	(* ----------------------------------------------------------------------------
	Const name  : FSM_EVENT_ARRAY_MAX
	Description : Max event array index value in the FSM table
				  Must subtract 1 due to arrays starting at 0
	Notes       : Used in FSM table definitions
	---------------------------------------------------------------------------- *)
	FSM_EVENT_ARRAY_MAX: INT := FSM_NUM_EVENTS - 1;
	
	(* ----------------------------------------------------------------------------
	Const name  : FSM_ACTIONS_ARRAY_MAX
	Description : Max actions array index value in the FSM table
				  next state entry is element 0 
	Notes       : Used in FSM table definitions
	---------------------------------------------------------------------------- *)
	FSM_ACTIONS_ARRAY_MAX: INT := FSM_NUM_EVENT_ACTIONS;

END_VAR

// (* FSM *)

//Run the Tri State Valve Finite State Machine Logic Block <JAISON>
m_TriStateValveControlFSM(xEnable:= xEnable, xError=> m_FsmError, errorNum=> m_FsmErrorNum);

//Set the current FSM State variable for testing the FSM state transitions <JAISON>
m_FsmCurrentState := m_TriStateValveControlFSM.FSM_GetCurrentState();

// Run the valve shift timer, the timer is enabled/disabled in the action handler. <JAISON>
//m_ShiftTimer(IN:= (m_TriStateValveControlFSM.FSM_GetCurrentState() = TriStateValveFsmState.FsmState_ValveShifting), PT:= ValveShiftTimeout);
m_ShiftTimer(PT:= ValveShiftTimeout);

// (* VALVE FEEDBACK *)
// Determine the current valve state (position) based on the feedback <JAISON>

// If the open and closed feedback are both TRUE or both FALSE the valve position is unknown
IF (Opened_Feedback = Closed_Feedback) THEN
	
	ValvePosition := TValveTriStatePosition.PosUnknown;
	
// If the opened feedback is TRUE and closed feedback is FALSE then the valve is opened
ELSIF ((Opened_Feedback) AND (NOT Closed_Feedback)) THEN
	
	ValvePosition := TValveTriStatePosition.PosOpened;
	
// If the closed feedback is TRUE and the open feedback is FALSE then the valve is closed
ELSIF ((Closed_Feedback) AND (NOT Opened_Feedback)) THEN
	
	ValvePosition := TValveTriStatePosition.PosClosed;
	
END_IF

// (* EVENT TRIGGERS *)

// Valve enabled trigger, basic FSM Event with no user parameters <JAISON>
m_EnableTrigger(CLK:= xEnable);
IF (m_EnableTrigger.Q)THEN
	//  FSM Reset needs to be called outside of the Action Handler routine. 
	//	Reset the FSM before sending the enable event. <JAISON>
	m_TriStateValveControlFSM.FSM_Reset();
	m_TriStateValveControlFSM.FSM_ProcessEvent(event:= TriStateValveFsmEvent.FsmEvent_ValveEnable);
END_IF

// Valve disabled trigger, basic FSM Event with no user parameters <JAISON>
m_DisableTrigger(CLK:= xEnable);
IF (m_DisableTrigger.Q)THEN
	m_TriStateValveControlFSM.FSM_ProcessEvent(event:= TriStateValveFsmEvent.FsmEvent_ValveDisable);
END_IF

// Valve shift timeout expired event trigger, basic FSM Event with no user parameters <JAISON>
m_ShiftTimeoutTrigger(CLK:= m_ShiftTimer.Q);
IF (m_ShiftTimeoutTrigger.Q) THEN
	m_TriStateValveControlFSM.FSM_ProcessEvent(event:= TriStateValveFsmEvent.FsmEvent_ValveShiftTimerExpired);
END_IF

// Valve opened event trigger, basic FSM Event with no user parameters <JAISON>
m_OpenedTrigger(CLK:= (ValvePosition = TValveTriStatePosition.PosOpened) AND (m_ValveCmdPosition = TValveTriStatePosition.PosOpened));
IF (m_OpenedTrigger.Q) THEN
	m_TriStateValveControlFSM.FSM_ProcessEvent(event:= TriStateValveFsmEvent.FsmEvent_ValveOpened);
END_IF

// Valve closed event trigger, basic FSM Event with no user parameters <JAISON>
m_ClosedTrigger(CLK:= (ValvePosition = TValveTriStatePosition.PosClosed) AND (m_ValveCmdPosition = TValveTriStatePosition.PosClosed));
IF (m_ClosedTrigger.Q) THEN
	m_TriStateValveControlFSM.FSM_ProcessEvent(event:= TriStateValveFsmEvent.FsmEvent_ValveClosed);
END_IF

// Valve position mismatch event trigger, basic FSM Event with no user parameters <JAISON>
// <Note: Ensure the cmd position is valid before sending event, this means valve has been shifted AT LEAST once.> <JAISON>
m_PositionMismatchTrigger(CLK:= ((m_ValveCmdPosition <> ValvePosition) AND ((m_ValveCmdPosition = TValveTriStatePosition.PosOpened) OR (m_ValveCmdPosition = TValveTriStatePosition.PosClosed))));
IF (m_PositionMismatchTrigger.Q) THEN
	m_TriStateValveControlFSM.FSM_ProcessEvent(event:= TriStateValveFsmEvent.FsmEvent_ValvePositionMismatch);
END_IF

(* ---------------------------------------------------------------------------
Func name   : 	CloseValve
Description : 	Sends an valve close event the the FSM 
				if the block is Enabled.
Inputs      :	None
Returns     : 	None
Notes       : 	This method should be triggered by an event 
				and not called cyclically to prevent flooding 
				the FSM event Queue.
--------------------------------------------------------------------------- *)

METHOD CloseValve : BOOL
VAR_INPUT
END_VAR
// Send the valve open event if the valve is enabled
IF xEnable THEN
	
	// Reset the valve shift timeout timer
	m_ShiftTimer(IN:= FALSE);
		
	// Clear the shifting error output
	ShiftingError := FALSE;

	m_TriStateValveControlFSM.FSM_ProcessEvent(event:= TriStateValveFsmEvent.FsmEvent_ValveClose);
	
END_IF
END_METHOD

(* ---------------------------------------------------------------------------
Func name   : 	ExecuteAction
Description : 	This method is a standardized handler for
				each action generated by the FSM
Inputs      :	p_FSM			-	pointer to the instantiation of the FSM object
				currentAction	-	current FSM action being processed
				currentEvent	-	current FSM event being processed
Returns     : 	BOOL			- 	result of action function (returning true means change state)
Notes       : 	The approach of using an interface enables the user 
				of the FSM to define and handle actions based 
				on their design and implementation.
				
				Return TRUE to change state, FALSE to remain in 
				the same state, unless the FSM has the alwaysChangeState
				set to TRUE, then it will change state regardless 
				of action handler return.
				
				If a conditional state is to be used this action handler
				routuine is responsible for setting the conditionalState 
				value using the FSM_SetConditionalState() function.
--------------------------------------------------------------------------- *)

METHOD ExecuteAction : BOOL
VAR_INPUT
	p_FSM			: POINTER TO fb_FSM;			// Pointer to the instantiation of the FSM object
	currentAction	: TFsmAction;					// Current FSM action being processed
	currentEvent	: TFsmEventDesc;				// Current FSM event being processed
END_VAR
VAR_OUTPUT

END_VAR
VAR

END_VAR
CASE currentAction OF
	
	TriStateValveFsmAction.FsmAction_None:
		
		// DO ACTION NONE
			
		// This would be a good place to simply log that the event occured. <JAISON>
			
		// RETURN TRUE
		ExecuteAction := TRUE;
	
	TriStateValveFsmAction.FsmAction_ValveEnabled:
	
		// DO ACTION VALVE ENABLED

		// Disable the actuator outputs
		Open_Actuator := FALSE;	
		Close_Actuator := FALSE;

		// Clear the shifting error to FALSE
		ShiftingError := FALSE;

		// Reset the valve shift timer
		m_ShiftTimer(IN := FALSE);

		// Clear all event triggers to ensure all events are captured on startup
		// NOTE: DO NOT RESET ENABLE/DISABLE TRIGGERS <JAISON>
		m_OpenedTrigger(CLK:= FALSE);
		m_ClosedTrigger(CLK:= FALSE);
		m_PositionMismatchTrigger(CLK:= FALSE);
		m_ShiftTimeoutTrigger(CLK:= FALSE);

		// Shift the valve to the Initial Valve State
		CASE InitialValvePosition OF
			
			TValveTriStatePosition.PosOpened:
			
				OpenValve();
			
			TValveTriStatePosition.PosClosed:
			
				CloseValve();
				
		ELSE
		
			// Error - Retained valve position invalid  <MESSAGE>
			// Default to CLOSED <JAISON>
			CloseValve();
		
		END_CASE
		
		// RETURN TRUE
		ExecuteAction := TRUE;
		
	TriStateValveFsmAction.FsmAction_ValveDisabled:	

		// DO ACTION VALVE DISABLED
		
		// Disable the actuator outputs
		Open_Actuator := FALSE;	
		Close_Actuator := FALSE;
		
		// RETURN TRUE
		ExecuteAction := TRUE;
		
	TriStateValveFsmAction.FsmAction_ValveOpen:
		
		// DO ACTION VALVE OPEN
		
		// Enable the Open actuator and Disable the Close actuator
		Close_Actuator := FALSE;
		Open_Actuator := TRUE;
		
		// Set the desired valve position to OPEN
		m_ValveCmdPosition := TValveTriStatePosition.PosOpened;
		
		// Start the valve shift timeout timer
		m_ShiftTimer(IN:= TRUE);
		
		// RETURN TRUE
		ExecuteAction := TRUE;
			
	TriStateValveFsmAction.FsmAction_ValveClose:
		
		// DO ACTION VALVE CLOSE

		// Enable the Close actuator and Disable the Open actuator
		Open_Actuator := FALSE;
		Close_Actuator := TRUE;
		
		// Set the desired valve position to CLOSE
		m_ValveCmdPosition := TValveTriStatePosition.PosClosed;
		
		// Start the valve shift timeout timer
		m_ShiftTimer(IN:= TRUE);
		
		// RETURN TRUE
		ExecuteAction := TRUE;
			
	TriStateValveFsmAction.FsmAction_ValveOpened:
		
		// DO ACTION VALVE OPENED
		
		// Disable both the Open and Close actuators
		Open_Actuator := FALSE;
		Close_Actuator := FALSE;
		
		// Clear the shifting error output
		ShiftingError := FALSE;
		
		// Stop the valve shift timeout timer
		m_ShiftTimer(IN:= FALSE);
		
		// RETURN TRUE
		ExecuteAction := TRUE;
			
	TriStateValveFsmAction.FsmAction_ValveClosed:
		
		// DO ACTION VALVE CLOSED
			
		// Disable both the Open and Close actuators
		Open_Actuator := FALSE;
		Close_Actuator := FALSE;
		
		// Clear the shifting error output
		ShiftingError := FALSE;
		
		// Stop the valve shift timeout timer
		m_ShiftTimer(IN:= FALSE);
		
		// RETURN TRUE
		ExecuteAction := TRUE;
			
	TriStateValveFsmAction.FsmAction_ValveShiftTimerExpired:
		
		// DO ACTION VALVE SHIFT TIMER EXPIRED
	
		// Set the shifting error output
		ShiftingError := TRUE;
				
		// RETURN TRUE
		ExecuteAction := TRUE;
		
	TriStateValveFsmAction.FsmAction_ValvePositionMismatch:
		
		// DO ACTION VALVE POSITION MISMATCH
		
		CASE m_ValveCmdPosition OF
			TValveTriStatePosition.PosOpened:
			
				// If the desired valve position is to be opened and the valve drifted then activate the open command again.
				p_FSM^.FSM_ProcessEvent(event:= TriStateValveFsmEvent.FsmEvent_ValveOpen);
			
			TValveTriStatePosition.PosClosed:
			
				// If the desired valve position is to be closed and the valve drifted then activate the close command again.
				p_FSM^.FSM_ProcessEvent(event:= TriStateValveFsmEvent.FsmEvent_ValveClose);
			
			ELSE
				
				// Error - Desired position unknown - Should not happen
				// NOTE: 	This will HALT the FSM when it FAILS which might not be the desired behavior.
				//			It is NOT necessary to halt the FSM, instead an unexpected event might just
				//			place the FSM into an error state which will allow actions to be ran. <JAISON>
				p_FSM^.FSM_ASSERT(FALSE, TFsmError.FSM_INVALID_EVENT_ERROR);
				
		END_CASE
		
		// RETURN TRUE
		ExecuteAction := TRUE;
			
	FSM_ACTION_UNEXPECTED_EVENT:
		
		// DO ACTION UNEXPECTED EVENT
		
		// ERROR TRAP - UNKNOWN ACTION
		// NOTE: 	This will HALT the FSM when it FAILS which is likely advisable here because
		//			this is a critical design time error.  All actions need to be defined, even
		//			if they simply log an event occured. <JAISON>
		p_FSM^.FSM_ASSERT(FALSE, TFsmError.FSM_INVALID_ACTION);
		
		// RETURN FALSE
		ExecuteAction := FALSE;
		
	FSM_ACTION_ERROR_EVENT:
	
		// DO ACTION ERROR EVENT
		
		// This action is executed when an FSM ASSERT Fails and the FSM is transitioning to the defined error state. <JAISON>
		
		// Automatically Reset the Valve / FSM by toggling the enable which will force the FSM to reset to Valve Off state
		m_EnableTrigger(CLK:= FALSE);
		
		// RETURN FALSE - This is irrelevant because the FSM will automatically transition to the error state.
		ExecuteAction := FALSE;
			
ELSE
		
	// ERROR TRAP - UNKNOWN ACTION
	// NOTE: 	This will HALT the FSM when it FAILS which is likely advisable here because
	//			this is a critical design time error.  All actions need to be defined, even
	//			if they simply log an event occured. <JAISON>
	p_FSM^.FSM_ASSERT(FALSE, TFsmError.FSM_INVALID_ACTION);
		
	// RETURN FALSE
	ExecuteAction := FALSE;
		
END_CASE;

m_FsmLastEvent := currentEvent.event;
m_FsmLastAction := currentAction;
m_FsmLastState := p_FSM^.FSM_GetPreviousState();
END_METHOD

(* ---------------------------------------------------------------------------
Func name   : 	FB_exit
Description : 	Destructor
Inputs      :	None
Returns     : 	None
Notes       : 	
--------------------------------------------------------------------------- *)

METHOD FB_exit : BOOL
VAR_INPUT
	bInCopyCode : BOOL; // if TRUE, the exit method is called for exiting an instance that is copied afterwards (online change)
END_VAR
// Do nothing
END_METHOD

(* ---------------------------------------------------------------------------
Func name   : 	FB_init
Description : 	Constructor
Inputs      :	None
Returns     : 	None
Notes       : 	
--------------------------------------------------------------------------- *)

METHOD FB_init : BOOL
VAR_INPUT
	bInitRetains 		: BOOL; 				// if TRUE, the retain variables are initialized (warm start / cold start)
    bInCopyCode  		: BOOL; 				// if TRUE, the instance afterwards gets moved into the copy code (online change)
END_VAR
// Set the FSM error state
// Technically this valve does NOT use the error state as it just resets itself 
// on transition to this state, however it is a good practice to have and will
// be useful for other state machines. <JAISON>
m_TriStateValveControlFSM.FSM_SetErrorState(TriStateValveFsmState.FsmState_Error);

// Clear all event triggers to ensure all events are captured on startup
m_EnableTrigger(CLK:= FALSE);
m_DisableTrigger(CLK:= FALSE);
m_OpenedTrigger(CLK:= FALSE);
m_ClosedTrigger(CLK:= FALSE);
m_PositionMismatchTrigger(CLK:= FALSE);
m_ShiftTimeoutTrigger(CLK:= FALSE);

// Initialize the default valve cmd state to unknown as this will be properly set during the valve enable. <JAISON>
m_ValveCmdPosition := TValveTriStatePosition.PosUnknown;

// Disable the actuator outputs
Open_Actuator := FALSE;	
Close_Actuator := FALSE;

// Initialize the shifting error to FALSE
ShiftingError := FALSE;
END_METHOD

(* ---------------------------------------------------------------------------
Func name   : 	OpenValve
Description : 	Sends an valve open event the the FSM 
				if the block is Enabled.
Inputs      :	None
Returns     : 	None
Notes       : 	This method should be triggered by an event 
				and not called cyclically to prevent flooding 
				the FSM event Queue.
--------------------------------------------------------------------------- *)

METHOD OpenValve
VAR_INPUT
END_VAR
// Send the valve open event if the valve is enabled
IF xEnable THEN

	// Reset the valve shift timeout timer
	m_ShiftTimer(IN:= FALSE);
		
	// Clear the shifting error output
	ShiftingError := FALSE;	

	m_TriStateValveControlFSM.FSM_ProcessEvent(event:= TriStateValveFsmEvent.FsmEvent_ValveOpen);
	
END_IF
END_METHOD

END_FUNCTION_BLOCK

// 20 Program Organization Units/Equipment Functions/TriStateValve/fb_DigitalFeedbackDualActionValve
(*AUTHOR:			Ryan Herdian*)
(*DATE:				July 30, 2020*)
(*DESCRIPTION: 		This function block provides the functionality for a Tri-State dual action valve which
					has digital boolean Open/Close feedback.  This valve is controlled by output
					boolean Open/Close solenoid and motor.*)

(*NOTES:			Operation of the valve are to follow
					To Open:
					-	Energize both solenoid and motor output at the same time. Until open. 
					-	Leave about 5 seconds after in position
					-	Remove power
					
					To Close:
					-	Energize the motor output only until close
					-	Leave about 5 seconds
					-	Remove power
					
					Currently, this function block is intended for
					- Emerson Damcos LPU-D
*)

(*UPDATE: 			March. 23 2021 - Jaison Schaab

					Code Is fully tested and functional.				
*)

(*UPDATE: 			March. 18 2021 - Jaison Schaab

					Code Ported from Wago.
					
					Code has NOT Yet been tested.
*)
	
(*UPDATE: 			September. 3 2020 - Jaison Schaab

					Added a "IsShifting" method for use in the control class development to detect when valve is shifting.
*)
					
(*UPDATE: 			September. 1 2020 - Jaison Schaab

					Added a "IsShiftingError" method for use in the control class development to detect valve shift error.
					
					Moved the setting of the outputs to occur through triggers rather than in the methods.  This was because
					during testing of the suction control class I noticed that the valves would not initially shift the their
					default position on startup; which is a massive concern.
*)

FUNCTION_BLOCK fb_DigitalFeedbackDualActionValve
VAR_INPUT
	xEnable						: BOOL;						// Enable inputs and valve operation
	OpenCommand					: BOOL;						// Open valve command input
	CloseCommand				: BOOL;						// Close valve command input
	InitialValvePosition		: TValveTriStatePosition;	// Position the valve will shift to when enabled (To be retianed if desired outside this block)
	OpenedFeedback				: BOOL;						// Digital feedback (TRUE = valve OPENED)
	ClosedFeedback				: BOOL;						// Digital feedback (TRUE = valve CLOSED)
	ValveShiftTimeout			: TIME;						// Valve shift timout value
	ValveOutputDisableTime		: TIME;						// Time to disable the output after shifting 
END_VAR
VAR_OUTPUT
	ValvePosition				: TValveTriStatePosition;	// Current valve position	(0 = closed, 1 = open)
	SolenoidEnergized			: BOOL;								// Solenoid energized (TRUE to OPEN valve together with Motor)
	MotorEnergized				: BOOL;								// Motor energized (TRUE to OPEN valve together with Solenoid)
END_VAR
VAR
	(* TriState Valve Function Block *)	

	m_TriStateValve				: fb_TriStateValve;			// Tri-State valve common control with state machine
	
	(* Valve Status *)	
	m_OpenedFeedback			: BOOL;						// Internal valve opened feedback
	m_ClosedFeedback			: BOOL;						// Internal valve closed feedback
	
	m_ValveShiftError			: BOOL;						// Valve shift timeout error flag
	
	(* Valve Internal Command *)
	m_OpenActuator				: BOOL;						// Internal Valve open actuator (TRUE to OPEN valve)
	m_CloseActuator				: BOOL;						// Internal Valve close actuator (TRUE to CLOSE valve)
	
	(* Alarms *)
	m_ValveShiftTimeout			: fb_AlarmMonitor;			// Alarm monitor for valve shift timeout error
	
	(* Event Triggers *)	

	m_EnableTrigger				: R_TRIG;					// Valve enabled trigger
	m_DisableTrigger			: F_TRIG;					// Valve disabled trigger
	m_OpenTrigger				: R_TRIG;					// Valve open trigger
	m_CloseTrigger				: R_TRIG;					// Valve close trigger
	m_ValveShiftErrorTrigger	: R_TRIG;					// Valve shift error trigger
	
	m_SetOpenActuatorTrigger	: R_TRIG;					// Set open actuator trigger
	m_SetCloseActuatorTrigger	: R_TRIG;					// Set close actuator trigger
	
	m_DisableOutputTrigger		: R_TRIG;					// Disable output trigger
	
	
	// ---- move this to the appropriate section
	//m_ValveShifted				: BOOL;
	// ----
	
	(* TIMER *)
	m_ValveShiftedTimer			: TON;
	
END_VAR

// Run the common TriState Valve function block which manages the state machine
m_TriStateValve(	xEnable					:= xEnable, 
					InitialValvePosition	:= InitialValvePosition,
					Opened_Feedback			:= m_OpenedFeedback, 
					Closed_Feedback			:= m_ClosedFeedback, 
					ValveShiftTimeout		:= ValveShiftTimeout,
					ValvePosition			=> ValvePosition, 
					Open_Actuator			=> m_OpenActuator, 
					Close_Actuator			=> m_CloseActuator, 
					ShiftingError			=> m_ValveShiftError);
					

(* TIMER *)
m_ValveShiftedTimer(IN:= IsOpened() OR IsClosed(), PT:= ValveOutputDisableTime);


// (* EVENT TRIGGERS *)

// Valve enabled trigger
m_EnableTrigger(CLK:= xEnable);
IF (m_EnableTrigger.Q)THEN
	
	// De-energized the Solenoid and Motor
	SolenoidEnergized := FALSE;
	MotorEnergized := FALSE;

	// Disable the internal actuator outputs
	m_OpenActuator := FALSE;	
	m_CloseActuator := FALSE;

	// Clear all event triggers to ensure all events are captured on startup
	// NOTE: DO NOT RESET ENABLE/DISABLE TRIGGERS
	m_OpenTrigger(CLK:= FALSE);
	m_CloseTrigger(CLK:= FALSE);
	
	m_ValveShiftErrorTrigger(CLK:= FALSE);
	
	m_SetOpenActuatorTrigger(CLK:= FALSE);
	m_SetCloseActuatorTrigger(CLK:= FALSE);
	
END_IF

// Valve disabled trigger
m_DisableTrigger(CLK:= xEnable);
IF (m_DisableTrigger.Q)THEN
	// Disable the alarm monitor
	m_ValveShiftTimeout.DisableLimit();
END_IF

// Open valve command event trigger
m_OpenTrigger(CLK:= OpenCommand);
IF (m_OpenTrigger.Q) THEN	
	OpenValve();	
END_IF

// Close valve command event trigger
m_CloseTrigger(CLK:= CloseCommand);
IF (m_CloseTrigger.Q) THEN
	CloseValve();		
END_IF

// Valve shift error event trigger
m_ValveShiftErrorTrigger(CLK:= m_ValveShiftError);
IF (m_ValveShiftErrorTrigger.Q) THEN
	// Reset the open/close actuator triggers to reissue the last command outputs
	m_SetOpenActuatorTrigger(CLK:= FALSE);
	m_SetCloseActuatorTrigger(CLK:= FALSE);
END_IF

// Open acutator trigger
m_SetOpenActuatorTrigger(CLK:= m_OpenActuator);
IF (m_SetOpenActuatorTrigger.Q) THEN
	SolenoidEnergized	:= TRUE;
	MotorEnergized		:= TRUE;
END_IF

// Close actuator trigger
m_SetCloseActuatorTrigger(CLK:= m_CloseActuator);
IF (m_SetCloseActuatorTrigger.Q) THEN
	MotorEnergized 		:= TRUE;
	SolenoidEnergized 	:= FALSE;		
END_IF
	
// Disable Output Trigger
m_DisableOutputTrigger(CLK:= m_ValveShiftError OR m_ValveShiftedTimer.Q);
IF (m_DisableOutputTrigger.Q)THEN	
	// De-energized the Solenoid and Motor
	SolenoidEnergized 	:= FALSE;
	MotorEnergized 		:= FALSE;	
END_IF


// (* VALVE FEEDBACK *)

// Decode the valve feedback
m_OpenedFeedback := OpenedFeedback;
m_ClosedFeedback := ClosedFeedback;


// Run the Alarm Monitors
m_ValveShiftTimeout.MonitorBool(value:= m_ValveShiftError);

(* ---------------------------------------------------------------------------
Func name   : 	CloseValve
Description : 	Sends an valve close event the the Tri-State valve if the block is Enabled.
				De-energize the Solenoid and Energize the Motor to close the valve if the
				valve has not already in the closed position.
Inputs      :	None
Returns     : 	None
Notes       : 	This method should be triggered by an event 
				and not called cyclically to prevent flooding 
				the FSM event Queue.
--------------------------------------------------------------------------- *)

METHOD CloseValve : BOOL
VAR_INPUT
END_VAR
// Send CLOSE command to Tri-State Valve FSM if the valve is enabled
IF xEnable THEN
	m_TriStateValve.CloseValve();	
END_IF
END_METHOD

(* ---------------------------------------------------------------------------
Func name   : 	FB_exit
Description : 	Destructor
Inputs      :	None
Returns     : 	None
Notes       : 	
--------------------------------------------------------------------------- *)

METHOD FB_exit : BOOL
VAR_INPUT
	bInCopyCode : BOOL; // if TRUE, the exit method is called for exiting an instance that is copied afterwards (online change)
END_VAR
// Do Nothing
END_METHOD

(* ---------------------------------------------------------------------------
Func name   : 	FB_init
Description : 	Constructor
Inputs      :	None
Returns     : 	None
Notes       : 	
--------------------------------------------------------------------------- *)

METHOD FB_init : BOOL
VAR_INPUT
	bInitRetains 		: BOOL; 				// if TRUE, the retain variables are initialized (warm start / cold start)
    bInCopyCode  		: BOOL; 				// if TRUE, the instance afterwards gets moved into the copy code (online change)
END_VAR
// Disable the solenoid and motor outputs
SolenoidEnergized := FALSE;
MotorEnergized := FALSE;

// Disable the actuator outputs
m_OpenActuator := FALSE;	
m_CloseActuator := FALSE;

// Clear all event triggers to ensure all events are captured on startup
m_EnableTrigger(CLK:= FALSE);
m_DisableTrigger(CLK:= FALSE);
m_OpenTrigger(CLK:= FALSE);
m_CloseTrigger(CLK:= FALSE);
m_ValveShiftErrorTrigger(CLK:= FALSE);
m_SetOpenActuatorTrigger(CLK:= FALSE);
m_SetCloseActuatorTrigger(CLK:= FALSE);
END_METHOD

(* ---------------------------------------------------------------------------
Func name   : 	InitAlarms
Description : 	Initializes the alarm monitors for the valve.
Inputs      :	devId	:	Device Id used for alarm integration
Returns     : 	None
Notes       : 	
--------------------------------------------------------------------------- *)

METHOD InitAlarms
VAR_INPUT
	devId	: UDeviceId;	// Device Id used for alarm integration
END_VAR
// Initialize the alarm monitors and set their limits
m_ValveShiftTimeout.InitAlarm( code:= f_AlarmCode( devId, f_FaultCode(TFaultPriority.Warning, TFaultCondition.TimeOut)), 
														  alarmType:= TAlarmMonitorType.upper_limit, 
														  delayTime:= T#1S);
m_ValveShiftTimeout.SetLimitBool(on:= TRUE, off:= FALSE);
m_ValveShiftTimeout.EnableLimit();
END_METHOD

(* ---------------------------------------------------------------------------
Func name   : 	IsClosed
Description : 	Polls valve for its closed status.
Inputs      :	None
Returns     : 	BOOL	-	TRUE is valve Closed, FALSE otherwise
Notes       : 	
--------------------------------------------------------------------------- *)

METHOD IsClosed : BOOL
VAR_INPUT
END_VAR
IsClosed := m_ClosedFeedback;
END_METHOD

(* ---------------------------------------------------------------------------
Func name   : 	IsOpened
Description : 	Polls valve for its opened status.
Inputs      :	None
Returns     : 	BOOL	-	TRUE is valve Opened, FALSE otherwise
Notes       : 	
--------------------------------------------------------------------------- *)

METHOD IsOpened : BOOL
VAR_INPUT
END_VAR
IsOpened := m_OpenedFeedback;
END_METHOD

(* ---------------------------------------------------------------------------
Func name   : 	IsShifting
Description : 	Polls valve for its shifting status.
Inputs      :	None
Returns     : 	BOOL	-	TRUE is valve is shifting, FALSE otherwise
Notes       : 	
--------------------------------------------------------------------------- *)

METHOD IsShifting : BOOL
VAR_INPUT
END_VAR
IF (ValvePosition = TValveTriStatePosition.PosUnknown) THEN
	IsShifting := TRUE;
ELSE
	IsShifting := FALSE;
END_IF
END_METHOD

(* ---------------------------------------------------------------------------
Func name   : 	IsShiftingError
Description : 	Polls valve for its shifting error status.
Inputs      :	None
Returns     : 	BOOL	-	TRUE is valve shift error, FALSE otherwise
Notes       : 	
--------------------------------------------------------------------------- *)

METHOD IsShiftingError : BOOL
VAR_INPUT
END_VAR
IsShiftingError	:= m_ValveShiftError;
END_METHOD

(* ---------------------------------------------------------------------------
Func name   : 	OpenValve
Description : 	Sends a valve open event the the Tri-State valve if the block is Enabled.
				Energize the Solenoid and Motor to open the valve if the valve has not 
				already in the opened position.
Inputs      :	None
Returns     : 	None
Notes       : 	This method should be triggered by an event 
				and not called cyclically to prevent flooding 
				the FSM event Queue.
--------------------------------------------------------------------------- *)

METHOD OpenValve : BOOL
VAR_INPUT
END_VAR
// Send OPEN command to Tri-State Valve FSM if the valve is enabled
IF xEnable THEN
	m_TriStateValve.OpenValve();	
END_IF
END_METHOD

END_FUNCTION_BLOCK

// 20 Program Organization Units/Equipment Functions/TriStateValve/fb_DigitalFeedbackSingleActionValve
(*AUTHOR:			Ryan Herdian*)
(*DATE:				August 04, 2020*)
(*DESCRIPTION: 		This function block provides the functionality for a Tri-State single action valve which
					has digital boolean Open/Close feedback.  This valve is controlled by output
					boolean Open/Close solenoid and motor.*)

(*NOTES:			Operation of the valve are to follow
					To Open:
					-	Energize both solenoid and motor output at the same time. Until open. 
					-	Leave power on / energized
					
					To Close:
					-	De-Energize both the solenoid motor output
					
					Currently, this function block is intended for
					- Emerson Damcos LPU-S
*)

(*UPDATE: 			March. 23 2021 - Jaison Schaab

					Code Is fully tested and functional.				
*)

(*UPDATE: 			March. 18 2021 - Jaison Schaab

					Code Ported from Wago.
					
					Code has NOT Yet been tested.
*)
	
(*UPDATE: 			September. 3 2020 - Jaison Schaab

					Added a "IsShifting" method for use in the control class development to detect when valve is shifting.
*)
					
(*UPDATE: 			September. 1 2020 - Jaison Schaab

					Added a "IsShiftingError" method for use in the control class development to detect valve shift error.
					
					Moved the setting of the outputs to occur through triggers rather than in the methods.  This was because
					during testing of the suction control class I noticed that the valves would not initially shift the their
					default position on startup; which is a massive concern.
*)

FUNCTION_BLOCK fb_DigitalFeedbackSingleActionValve
VAR_INPUT
	xEnable						: BOOL;						// Enable inputs and valve operation
	OpenCommand					: BOOL;						// Open valve command input
	CloseCommand				: BOOL;						// Close valve command input
	InitialValvePosition		: TValveTriStatePosition;	// Position the valve will shift to when enabled (To be retianed if desired outside this block)
	OpenedFeedback				: BOOL;						// Digital feedback (TRUE = valve OPENED)
	ClosedFeedback				: BOOL;						// Digital feedback (TRUE = valve CLOSED)
	ValveShiftTimeout			: TIME;						// Valve shift timout value
END_VAR
VAR_OUTPUT
	ValvePosition				: TValveTriStatePosition;	// Current valve position	(0 = closed, 1 = open)
	SolenoidEnergized			: BOOL;								// Solenoid energized (TRUE to OPEN valve together with Motor)
	MotorEnergized				: BOOL;								// Motor energized (TRUE to OPEN valve together with Solenoid)
END_VAR
VAR
	(* TriState Valve Function Block *)	

	m_TriStateValve				: fb_TriStateValve;			// Tri-State valve common control with state machine
	
	(* Valve Status *)	
	m_OpenedFeedback			: BOOL;						// Internal valve opened feedback
	m_ClosedFeedback			: BOOL;						// Internal valve closed feedback
	
	m_ValveShiftError			: BOOL;						// Valve shift timeout error flag
	
	(* Valve Internal Command *)
	m_OpenActuator				: BOOL;						// Internal Valve open actuator (TRUE to OPEN valve)
	m_CloseActuator				: BOOL;						// Internal Valve close actuator (TRUE to CLOSE valve)
	
	(* Alarms *)
	m_ValveShiftTimeout			: fb_AlarmMonitor;			// Alarm monitor for valve shift timeout error
	
	(* Event Triggers *)	

	m_EnableTrigger				: R_TRIG;					// Valve enabled trigger
	m_DisableTrigger			: F_TRIG;					// Valve disabled trigger
	m_OpenTrigger				: R_TRIG;					// Valve open trigger
	m_CloseTrigger				: R_TRIG;					// Valve close trigger
	m_ValveShiftErrorTrigger	: R_TRIG;					// Valve shift error trigger
	
	m_SetOpenActuatorTrigger	: R_TRIG;					// Set open actuator trigger
	m_SetCloseActuatorTrigger	: R_TRIG;					// Set close actuator trigger
	
	m_DisableOutputTrigger		: R_TRIG;					// Disable output trigger
	
END_VAR

// Run the common TriState Valve function block which manages the state machine
m_TriStateValve(	xEnable					:= xEnable, 
					InitialValvePosition	:= InitialValvePosition,
					Opened_Feedback			:= m_OpenedFeedback, 
					Closed_Feedback			:= m_ClosedFeedback, 
					ValveShiftTimeout		:= ValveShiftTimeout,
					ValvePosition			=> ValvePosition, 
					Open_Actuator			=> m_OpenActuator, 
					Close_Actuator			=> m_CloseActuator, 
					ShiftingError			=> m_ValveShiftError);


// (* EVENT TRIGGERS *)

// Valve enabled trigger
m_EnableTrigger(CLK:= xEnable);
IF (m_EnableTrigger.Q)THEN
	
	// De-energized the Solenoid and Motor
	SolenoidEnergized := FALSE;
	MotorEnergized := FALSE;

	// Disable the internal actuator outputs
	m_OpenActuator := FALSE;	
	m_CloseActuator := FALSE;

	// Clear all event triggers to ensure all events are captured on startup
	// NOTE: DO NOT RESET ENABLE/DISABLE TRIGGERS
	m_OpenTrigger(CLK:= FALSE);
	m_CloseTrigger(CLK:= FALSE);
	
	m_ValveShiftErrorTrigger(CLK:= FALSE);
	
	m_SetOpenActuatorTrigger(CLK:= FALSE);
	m_SetCloseActuatorTrigger(CLK:= FALSE);
	
END_IF

// Valve disabled trigger
m_DisableTrigger(CLK:= xEnable);
IF (m_DisableTrigger.Q)THEN
	// Disable the alarm monitor
	m_ValveShiftTimeout.DisableLimit();
END_IF

// Open valve command event trigger
m_OpenTrigger(CLK:= OpenCommand);
IF (m_OpenTrigger.Q) THEN	
	OpenValve();	
END_IF

// Close valve command event trigger
m_CloseTrigger(CLK:= CloseCommand);
IF (m_CloseTrigger.Q) THEN
	CloseValve();		
END_IF

// Valve shift error event trigger
m_ValveShiftErrorTrigger(CLK:= m_ValveShiftError);
IF (m_ValveShiftErrorTrigger.Q) THEN
	// Reset the open/close actuator triggers to reissue the last command outputs
	m_SetOpenActuatorTrigger(CLK:= FALSE);
	m_SetCloseActuatorTrigger(CLK:= FALSE);
END_IF

// Open acutator trigger
m_SetOpenActuatorTrigger(CLK:= m_OpenActuator);
IF (m_SetOpenActuatorTrigger.Q) THEN
	SolenoidEnergized	:= TRUE;
	MotorEnergized		:= TRUE;
END_IF

// Close actuator trigger
m_SetCloseActuatorTrigger(CLK:= m_CloseActuator);
IF (m_SetCloseActuatorTrigger.Q) THEN
	MotorEnergized 		:= FALSE;
	SolenoidEnergized 	:= FALSE;		
END_IF

// Disable Output Trigger
m_DisableOutputTrigger(CLK:= m_ValveShiftError);
IF (m_DisableOutputTrigger.Q)THEN	
	// De-energized the Solenoid and Motor
	SolenoidEnergized := FALSE;
	MotorEnergized := FALSE;	
END_IF


// (* VALVE FEEDBACK *)

// Decode the valve feedback
m_OpenedFeedback := OpenedFeedback;
m_ClosedFeedback := ClosedFeedback;


// Run the Alarm Monitors
m_ValveShiftTimeout.MonitorBool(value:= m_ValveShiftError);

(* ---------------------------------------------------------------------------
Func name   : 	CloseValve
Description : 	Sends a valve close event the the Tri-State valve if the block is Enabled.
				De-energize the Solenoid and the Motor to close the valve if the
				valve has not already in the closed position.
Inputs      :	None
Returns     : 	None
Notes       : 	This method should be triggered by an event 
				and not called cyclically to prevent flooding 
				the FSM event Queue.
--------------------------------------------------------------------------- *)

METHOD CloseValve : BOOL
VAR_INPUT
END_VAR
// Send CLOSE command to Tri-State Valve FSM if the valve is enabled
IF xEnable THEN
	m_TriStateValve.CloseValve();
END_IF
END_METHOD

(* ---------------------------------------------------------------------------
Func name   : 	FB_exit
Description : 	Destructor
Inputs      :	None
Returns     : 	None
Notes       : 	
--------------------------------------------------------------------------- *)

METHOD FB_exit : BOOL
VAR_INPUT
	bInCopyCode : BOOL; // if TRUE, the exit method is called for exiting an instance that is copied afterwards (online change)
END_VAR
// Do Nothing
END_METHOD

(* ---------------------------------------------------------------------------
Func name   : 	FB_init
Description : 	Constructor
Inputs      :	None
Returns     : 	None
Notes       : 	
--------------------------------------------------------------------------- *)

METHOD FB_init : BOOL
VAR_INPUT
	bInitRetains 		: BOOL; 				// if TRUE, the retain variables are initialized (warm start / cold start)
    bInCopyCode  		: BOOL; 				// if TRUE, the instance afterwards gets moved into the copy code (online change)
END_VAR
// Disable the solenoid and motor outputs
SolenoidEnergized := FALSE;
MotorEnergized := FALSE;

// Disable the actuator outputs
m_OpenActuator := FALSE;	
m_CloseActuator := FALSE;

// Clear all event triggers to ensure all events are captured on startup
m_EnableTrigger(CLK:= FALSE);
m_DisableTrigger(CLK:= FALSE);
m_OpenTrigger(CLK:= FALSE);
m_CloseTrigger(CLK:= FALSE);
m_ValveShiftErrorTrigger(CLK:= FALSE);
m_SetOpenActuatorTrigger(CLK:= FALSE);
m_SetCloseActuatorTrigger(CLK:= FALSE);
END_METHOD

(* ---------------------------------------------------------------------------
Func name   : 	InitAlarms
Description : 	Initializes the alarm monitors for the valve.
Inputs      :	devId	:	Device Id used for alarm integration
Returns     : 	None
Notes       : 	
--------------------------------------------------------------------------- *)

METHOD InitAlarms
VAR_INPUT
	devId	: UDeviceId;	// Device Id used for alarm integration
END_VAR
// Initialize the alarm monitors and set their limits
m_ValveShiftTimeout.InitAlarm( code:= f_AlarmCode( devId, f_FaultCode(TFaultPriority.Warning, TFaultCondition.TimeOut)), 
														  alarmType:= TAlarmMonitorType.upper_limit, 
														  delayTime:= T#1S);
m_ValveShiftTimeout.SetLimitBool(on:= TRUE, off:= FALSE);
m_ValveShiftTimeout.EnableLimit();
END_METHOD

(* ---------------------------------------------------------------------------
Func name   : 	IsClosed
Description : 	Polls valve for its closed status.
Inputs      :	None
Returns     : 	BOOL	-	TRUE is valve Closed, FALSE otherwise
Notes       : 	
--------------------------------------------------------------------------- *)

METHOD IsClosed : BOOL
VAR_INPUT
END_VAR
IsClosed := m_ClosedFeedback;
END_METHOD

(* ---------------------------------------------------------------------------
Func name   : 	IsOpened
Description : 	Polls valve for its opened status.
Inputs      :	None
Returns     : 	BOOL	-	TRUE is valve Opened, FALSE otherwise
Notes       : 	
--------------------------------------------------------------------------- *)

METHOD IsOpened : BOOL
VAR_INPUT
END_VAR
IsOpened := m_OpenedFeedback;
END_METHOD

(* ---------------------------------------------------------------------------
Func name   : 	IsShifting
Description : 	Polls valve for its shifting status.
Inputs      :	None
Returns     : 	BOOL	-	TRUE is valve is shifting, FALSE otherwise
Notes       : 	
--------------------------------------------------------------------------- *)

METHOD IsShifting : BOOL
VAR_INPUT
END_VAR
IF (ValvePosition = TValveTriStatePosition.PosUnknown) THEN
	IsShifting := TRUE;
ELSE
	IsShifting := FALSE;
END_IF
END_METHOD

(* ---------------------------------------------------------------------------
Func name   : 	IsShiftingError
Description : 	Polls valve for its shifting error status.
Inputs      :	None
Returns     : 	BOOL	-	TRUE is valve shift error, FALSE otherwise
Notes       : 	
--------------------------------------------------------------------------- *)

METHOD IsShiftingError : BOOL
VAR_INPUT
END_VAR
IsShiftingError	:= m_ValveShiftError;
END_METHOD

(* ---------------------------------------------------------------------------
Func name   : 	OpenValve
Description : 	Sends a valve open event the the Tri-State valve if the block is Enabled.
				Energize the Solenoid and Motor to open the valve if the valve has not 
				already in the opened position.
Inputs      :	None
Returns     : 	None
Notes       : 	This method should be triggered by an event 
				and not called cyclically to prevent flooding 
				the FSM event Queue.
--------------------------------------------------------------------------- *)

METHOD OpenValve : BOOL
VAR_INPUT
END_VAR
// Send OPEN command to Tri-State Valve FSM if the valve is enabled
IF xEnable THEN
	m_TriStateValve.OpenValve();
END_IF
END_METHOD

END_FUNCTION_BLOCK

// 20 Program Organization Units/Equipment Functions/TriStateValve/fb_DigitalFeedbackValve
(*AUTHOR:			Jaison Schaab*)
(*DATE:				March. 12 / 2020*)
(*DESCRIPTION: 		This function block provides the functionality for a Tri-State valve which
					has digital boolean Open/Close feedback.  This valve is controlled by output
					boolean Open/Close actuators.*)

(*UPDATE: 			March. 23 2021 - Jaison Schaab

					Code Is fully tested and functional.				
*)

(*UPDATE: 			March. 18 2021 - Jaison Schaab

					Code Ported from Wago.
					
					Code has NOT Yet been tested.
*)

(*UPDATE: 			September. 3 2020 - Jaison Schaab

					Added a "IsShifting" method for use in the control class development to detect when valve is shifting.
*)

(*UPDATE: 			September. 1 2020 - Jaison Schaab

					Added a "IsShiftingError" method for use in the control class development to detect valve shift error.
*)
					
(*UPDATE: 			April. 28 2020 - Jaison Schaab

					Added the InitAlarms function which now NEEDS to be called in order to properly hook up the alarm monitors.
					This method is required because codesys does NOT properly propogate the FB_Init information like constructors
					in C code, so it is impossible to pass down the devceId information.
*)

FUNCTION_BLOCK fb_DigitalFeedbackValve
VAR_INPUT
	xEnable						: BOOL;						// Enable inputs and valve operation
	OpenCommand					: BOOL;						// Open valve command input
	CloseCommand				: BOOL;						// Close valve command input
	InitialValvePosition		: TValveTriStatePosition;	// Position the valve will shift to when enabled (To be retianed if desired outside this block)
	OpenedFeedback				: BOOL;						// Digital feedback (TRUE = valve OPENED)
	ClosedFeedback				: BOOL;						// Digital feedback (TRUE = valve CLOSED)
	ValveShiftTimeout			: TIME;						// Valve shift timout value
END_VAR
VAR_OUTPUT
	ValvePosition				: TValveTriStatePosition;	// Current valve position	(0 = closed, 1 = open)
	OpenActuator				: BOOL;						// Valve open actuator (TRUE to OPEN valve)
	CloseActuator				: BOOL;						// Valve close actuator (TRUE to CLOSE valve)
END_VAR
VAR
	(* TriState Valve Function Block *)	

	m_TriStateValve				: fb_TriStateValve;			// Tri-State valve common control with state machine
	
	(* Valve Status *)	
	m_OpenedFeedback			: BOOL;						// Internal valve opened feedback
	m_ClosedFeedback			: BOOL;						// Internal valve closed feedback
	
	m_ValveShiftError			: BOOL;						// Valve shift timeout error flag
	
	(* Alarms *)
	m_ValveShiftTimeout			: fb_AlarmMonitor;			// Alarm monitor for valve shift timeout error
	
	(* Event Triggers *)	

	m_EnableTrigger				: R_TRIG;					// Valve enabled trigger
	m_DisableTrigger			: F_TRIG;					// Valve disabled trigger
	m_OpenTrigger				: R_TRIG;					// Valve open trigger
	m_CloseTrigger				: R_TRIG;					// Valve close trigger

END_VAR

// Run the common TriState Valve function block which manages the state machine
m_TriStateValve(	xEnable					:= xEnable, 
					InitialValvePosition	:= InitialValvePosition,
					Opened_Feedback			:= m_OpenedFeedback, 
					Closed_Feedback			:= m_ClosedFeedback, 
					ValveShiftTimeout		:= ValveShiftTimeout,
					ValvePosition			=> ValvePosition, 
					Open_Actuator			=> OpenActuator, 
					Close_Actuator			=> CloseActuator, 
					ShiftingError			=> m_ValveShiftError);

// (* EVENT TRIGGERS *)

// Valve enabled trigger
m_EnableTrigger(CLK:= xEnable);
IF (m_EnableTrigger.Q)THEN
	
	// Disable the actuator outputs
	OpenActuator := FALSE;	
	CloseActuator := FALSE;

	// Clear all event triggers to ensure all events are captured on startup
	// NOTE: DO NOT RESET ENABLE/DISABLE TRIGGERS <JAISON>
	m_OpenTrigger(CLK:= FALSE);
	m_CloseTrigger(CLK:= FALSE);
	
END_IF

// Valve disabled trigger
m_DisableTrigger(CLK:= xEnable);
IF (m_DisableTrigger.Q)THEN
	// Disable the alarm monitor
	m_ValveShiftTimeout.DisableLimit();
END_IF

// Open valve command event trigger <JAISON>
m_OpenTrigger(CLK:= OpenCommand);
IF (m_OpenTrigger.Q) THEN
	OpenValve();
END_IF

// Close valve command event trigger <JAISON>
m_CloseTrigger(CLK:= CloseCommand);
IF (m_CloseTrigger.Q) THEN
	CloseValve();
END_IF

// (* VALVE FEEDBACK *)

// Decode the valve feedback <JAISON>
m_OpenedFeedback := OpenedFeedback;
m_ClosedFeedback := ClosedFeedback;


// Run the Alarm Monitors <JAISON>
m_ValveShiftTimeout.MonitorBool(value:= m_ValveShiftError);

(* ---------------------------------------------------------------------------
Func name   : 	CloseValve
Description : 	Sends a valve close event the the Tri-State 
				valve if the block is Enabled.
Inputs      :	None
Returns     : 	None
Notes       : 	This method should be triggered by an event 
				and not called cyclically to prevent flooding 
				the FSM event Queue.
--------------------------------------------------------------------------- *)

METHOD CloseValve : BOOL
VAR_INPUT
END_VAR
// Send CLOSE command to Tri-State Valve FSM if the valve is enabled
IF xEnable THEN
	m_TriStateValve.CloseValve();
END_IF
END_METHOD

(* ---------------------------------------------------------------------------
Func name   : 	FB_exit
Description : 	Destructor
Inputs      :	None
Returns     : 	None
Notes       : 	
--------------------------------------------------------------------------- *)

METHOD FB_exit : BOOL
VAR_INPUT
	bInCopyCode : BOOL; // if TRUE, the exit method is called for exiting an instance that is copied afterwards (online change)
END_VAR
// Do Nothing
END_METHOD

(* ---------------------------------------------------------------------------
Func name   : 	FB_init
Description : 	Constructor
Inputs      :	None
Returns     : 	None
Notes       : 	
--------------------------------------------------------------------------- *)

METHOD FB_init : BOOL
VAR_INPUT
	bInitRetains 		: BOOL; 				// if TRUE, the retain variables are initialized (warm start / cold start)
    bInCopyCode  		: BOOL; 				// if TRUE, the instance afterwards gets moved into the copy code (online change)
END_VAR
// Disable the actuator outputs
OpenActuator := FALSE;	
CloseActuator := FALSE;

// Clear all event triggers to ensure all events are captured on startup
m_EnableTrigger(CLK:= FALSE);
m_DisableTrigger(CLK:= FALSE);
m_OpenTrigger(CLK:= FALSE);
m_CloseTrigger(CLK:= FALSE);
END_METHOD

(* ---------------------------------------------------------------------------
Func name   : 	InitAlarms
Description : 	Initializes the alarm monitors for the valve.
Inputs      :	devId	:	Device Id used for alarm integration
Returns     : 	None
Notes       : 	
--------------------------------------------------------------------------- *)

METHOD InitAlarms
VAR_INPUT
	devId	: UDeviceId;	// Device Id used for alarm integration
END_VAR
// Initialize the alarm monitors and set their limits
m_ValveShiftTimeout.InitAlarm(code:= f_AlarmCode(devId, f_FaultCode(TFaultPriority.Warning, TFaultCondition.TimeOut)), alarmType:= TAlarmMonitorType.upper_limit, delayTime:= T#1S);
m_ValveShiftTimeout.SetLimitBool(on:= TRUE, off:= FALSE);
m_ValveShiftTimeout.EnableLimit();
END_METHOD

(* ---------------------------------------------------------------------------
Func name   : 	IsClosed
Description : 	Polls valve for its closed status.
Inputs      :	None
Returns     : 	BOOL	-	TRUE is valve Closed, FALSE otherwise
Notes       : 	
--------------------------------------------------------------------------- *)

METHOD IsClosed : BOOL
VAR_INPUT
END_VAR
IsClosed := m_ClosedFeedback;
END_METHOD

(* ---------------------------------------------------------------------------
Func name   : 	IsOpened
Description : 	Polls valve for its opened status.
Inputs      :	None
Returns     : 	BOOL	-	TRUE is valve Opened, FALSE otherwise
Notes       : 	
--------------------------------------------------------------------------- *)

METHOD IsOpened : BOOL
VAR_INPUT
END_VAR
IsOpened := m_OpenedFeedback;
END_METHOD

(* ---------------------------------------------------------------------------
Func name   : 	IsShifting
Description : 	Polls valve for its shifting status.
Inputs      :	None
Returns     : 	BOOL	-	TRUE is valve is shifting, FALSE otherwise
Notes       : 	
--------------------------------------------------------------------------- *)

METHOD IsShifting : BOOL
VAR_INPUT
END_VAR
IF (ValvePosition = TValveTriStatePosition.PosUnknown) THEN
	IsShifting := TRUE;
ELSE
	IsShifting := FALSE;
END_IF
END_METHOD

(* ---------------------------------------------------------------------------
Func name   : 	IsShiftingError
Description : 	Polls valve for its shifting error status.
Inputs      :	None
Returns     : 	BOOL	-	TRUE is valve shift error, FALSE otherwise
Notes       : 	
--------------------------------------------------------------------------- *)

METHOD IsShiftingError : BOOL
VAR_INPUT
END_VAR
IsShiftingError	:= m_ValveShiftError;
END_METHOD

(* ---------------------------------------------------------------------------
Func name   : 	OpenValve
Description : 	Sends an valve open event the the Tri-State
				valve if the block is Enabled.
Inputs      :	None
Returns     : 	None
Notes       : 	This method should be triggered by an event 
				and not called cyclically to prevent flooding 
				the FSM event Queue.
--------------------------------------------------------------------------- *)

METHOD OpenValve : BOOL
VAR_INPUT
END_VAR
// Send OPEN command to Tri-State Valve FSM if the valve is enabled
IF xEnable THEN
	m_TriStateValve.OpenValve();
END_IF
END_METHOD

END_FUNCTION_BLOCK

// 20 Program Organization Units/Equipment Functions/TriStateValve/fb_NoFeedbackValve
(*AUTHOR:			Jaison Schaab*)
(*DATE:				March. 12 / 2020*)
(*DESCRIPTION: 		This function block provides the functionality for a Tri-State valve which
					has no feedback.  This valve is controlled by output boolean Open/Close 
					actuators.  The valve is automatically assumed shifted once ite actuated
					because there is no feedback.*)

(*UPDATE: 			March. 23 2021 - Jaison Schaab

					Code Is fully tested and functional.				
*)

(*UPDATE: 			March. 18 2021 - Jaison Schaab

					Code Ported from Wago.
					
					Code has NOT Yet been tested.
*)

(*UPDATE: 			September. 3 2020 - Jaison Schaab

					Added a "IsShifting" method for use in the control class development to detect when valve is shifting.
*)

(*UPDATE: 			September. 1 2020 - Jaison Schaab

					Added a "IsShiftingError" method for use in the control class development to detect valve shift error.
*)

FUNCTION_BLOCK fb_NoFeedbackValve
VAR_INPUT
	xEnable						: BOOL;						// Enable inputs and valve operation
	OpenCommand					: BOOL;						// Open valve command input
	CloseCommand				: BOOL;						// Close valve command input
	InitialValvePosition		: TValveTriStatePosition;	// Position the valve will shift to when enabled (To be retianed if desired outside this block)
END_VAR
VAR_OUTPUT
	ValvePosition				: TValveTriStatePosition;	// Current valve position	(0 = closed, 1 = open)
	OpenActuator				: BOOL;						// Valve open actuator (TRUE to OPEN valve)
	CloseActuator				: BOOL;						// Valve close actuator (TRUE to CLOSE valve)
END_VAR
VAR
	(* TriState Valve Function Block *)	

	m_TriStateValve				: fb_TriStateValve;			// Tri-State valve common control with state machine
	
	(* Valve Status *)	
	m_OpenedFeedback			: BOOL;						// Internal valve opened feedback
	m_ClosedFeedback			: BOOL;						// Internal valve closed feedback
	
	OpenBiStable				: RS;						// Triggers for valve opened feedback logic
	CloseBiStable				: RS;						// Triggers for valve closed feedback logic
	
	m_ValveShiftError			: BOOL;						// Valve shift timeout error flag
	
	(* Alarms *)
	
	// NONE
	
	(* Event Triggers *)	

	m_EnableTrigger				: R_TRIG;					// Valve enabled trigger
	m_DisableTrigger			: F_TRIG;					// Valve disabled trigger
	m_OpenTrigger				: R_TRIG;					// Valve open trigger
	m_CloseTrigger				: R_TRIG;					// Valve close trigger

END_VAR

// Run the common TriState Valve function block which manages the state machine
m_TriStateValve(	xEnable					:= xEnable, 
					InitialValvePosition	:= InitialValvePosition,
					Opened_Feedback			:= m_OpenedFeedback, 
					Closed_Feedback			:= m_ClosedFeedback, 
					ValveShiftTimeout		:= T#100S, // No shifting time without feedback, No error should be generated <JAISON>
					ValvePosition			=> ValvePosition, 
					Open_Actuator			=> OpenActuator, 
					Close_Actuator			=> CloseActuator, 
					ShiftingError			=> m_ValveShiftError);
					
// (* EVENT TRIGGERS *)

// Valve enabled trigger
m_EnableTrigger(CLK:= xEnable);
IF (m_EnableTrigger.Q)THEN
	
	// Disable the actuator outputs
	OpenActuator := FALSE;	
	CloseActuator := FALSE;

	// Clear all event triggers to ensure all events are captured on startup
	// NOTE: DO NOT RESET ENABLE/DISABLE TRIGGERS <JAISON>
	m_OpenTrigger(CLK:= FALSE);
	m_CloseTrigger(CLK:= FALSE);

END_IF

// Valve disabled trigger
m_DisableTrigger(CLK:= xEnable);
IF (m_DisableTrigger.Q)THEN
	// Do Nothing
END_IF

// Open valve command event trigger <JAISON>
m_OpenTrigger(CLK:= OpenCommand);
IF (m_OpenTrigger.Q) THEN
	OpenValve();
END_IF

// Close valve command event trigger <JAISON>
m_CloseTrigger(CLK:= CloseCommand);
IF (m_CloseTrigger.Q) THEN
	CloseValve();
END_IF

// (* VALVE FEEDBACK *)

// Decode the valve feedback.
// Because there is no actual feedback, simply assume the valve shifts
// when the actuator is set. <JAISON>
OpenBiStable(SET:= OpenActuator, RESET1:= CloseActuator, Q1=> m_OpenedFeedback);
CloseBiStable(SET:= CloseActuator, RESET1:= OpenActuator, Q1=> m_ClosedFeedback);

(* ---------------------------------------------------------------------------
Func name   : 	CloseValve
Description : 	Sends an valve close event the the Tri-State 
				valve if the block is Enabled.
Inputs      :	None
Returns     : 	None
Notes       : 	This method should be triggered by an event 
				and not called cyclically to prevent flooding 
				the FSM event Queue.
--------------------------------------------------------------------------- *)

METHOD CloseValve
VAR_INPUT
END_VAR
// Send CLOSE command to Tri-State Valve FSM if the valve is enabled
IF xEnable THEN
	m_TriStateValve.CloseValve();
END_IF
END_METHOD

(* ---------------------------------------------------------------------------
Func name   : 	FB_exit
Description : 	Destructor
Inputs      :	None
Returns     : 	None
Notes       : 	
--------------------------------------------------------------------------- *)

METHOD FB_exit : BOOL
VAR_INPUT
	bInCopyCode : BOOL; // if TRUE, the exit method is called for exiting an instance that is copied afterwards (online change)
END_VAR
// Do Nothing
END_METHOD

(* ---------------------------------------------------------------------------
Func name   : 	FB_init
Description : 	Constructor
Inputs      :	None
Returns     : 	None
Notes       : 	
--------------------------------------------------------------------------- *)

METHOD FB_init : BOOL
VAR_INPUT
	bInitRetains 		: BOOL; 				// if TRUE, the retain variables are initialized (warm start / cold start)
    bInCopyCode  		: BOOL; 				// if TRUE, the instance afterwards gets moved into the copy code (online change)
END_VAR
// Disable the actuator outputs
OpenActuator := FALSE;	
CloseActuator := FALSE;

// Clear all event triggers to ensure all events are captured on startup
m_EnableTrigger(CLK:= FALSE);
m_DisableTrigger(CLK:= FALSE);
m_OpenTrigger(CLK:= FALSE);
m_CloseTrigger(CLK:= FALSE);
END_METHOD

(* ---------------------------------------------------------------------------
Func name   : 	IsClosed
Description : 	Polls valve for its closed status.
Inputs      :	None
Returns     : 	BOOL	-	TRUE is valve Closed, FALSE otherwise
Notes       : 	
--------------------------------------------------------------------------- *)

METHOD IsClosed : BOOL
VAR_INPUT
END_VAR
IsClosed := m_ClosedFeedback;
END_METHOD

(* ---------------------------------------------------------------------------
Func name   : 	IsOpened
Description : 	Polls valve for its opened status.
Inputs      :	None
Returns     : 	BOOL	-	TRUE is valve Opened, FALSE otherwise
Notes       : 	
--------------------------------------------------------------------------- *)

METHOD IsOpened : BOOL
VAR_INPUT
END_VAR
IsOpened := m_OpenedFeedback;
END_METHOD

(* ---------------------------------------------------------------------------
Func name   : 	IsShifting
Description : 	Polls valve for its shifting status.
Inputs      :	None
Returns     : 	BOOL	-	TRUE is valve is shifting, FALSE otherwise
Notes       : 	
--------------------------------------------------------------------------- *)

METHOD IsShifting : BOOL
VAR_INPUT
END_VAR
IF (ValvePosition = TValveTriStatePosition.PosUnknown) THEN
	IsShifting := TRUE;
ELSE
	IsShifting := FALSE;
END_IF
END_METHOD

(* ---------------------------------------------------------------------------
Func name   : 	IsShiftingError
Description : 	Polls valve for its shifting error status.
Inputs      :	None
Returns     : 	BOOL	-	TRUE is valve shift error, FALSE otherwise
Notes       : 	
--------------------------------------------------------------------------- *)

METHOD IsShiftingError : BOOL
VAR_INPUT
END_VAR
IsShiftingError	:= m_ValveShiftError;
END_METHOD

(* ---------------------------------------------------------------------------
Func name   : 	OpenValve
Description : 	Sends an valve open event the the Tri-State
				valve if the block is Enabled.
Inputs      :	None
Returns     : 	None
Notes       : 	This method should be triggered by an event 
				and not called cyclically to prevent flooding 
				the FSM event Queue.
--------------------------------------------------------------------------- *)

METHOD OpenValve
VAR_INPUT
END_VAR
// Send OPEN command to Tri-State Valve FSM if the valve is enabled
IF xEnable THEN
	m_TriStateValve.OpenValve();
END_IF
END_METHOD

END_FUNCTION_BLOCK

// 20 Program Organization Units/Input-Output Functions/fb_AnalogOutputActuator
(*AUTHOR:			Graham Hunter*)
(*DATE:				October 28 / 2020*)
(*DESCRIPTION: 		This Function Block provides a base class for all analog output values.  
					The block converts a linear scaled 4 to 20 mA, 0 to 10V, or -10 to 10V signal to a linear scaled card count output value.
					
					Use the "AO_ChannelOutputs" data type to link the channel data from the physical I/O card. 
					Most of this functionality was duplicated from fb_Analog Transducer except the following Input and Outputs were switched:
 
 					// Card input (4 to 20mA, 0 to 10V, or -10V to 10V)
					m_iMinInput				: REAL;				// minimum commanded input (4.0 mA, 0V, or -10V )
					m_iMaxInput				: REAL;				// maximum commanded input (20.0 mA or 10V)

					// Card output (counts, -32768 to 32767)
					m_rMinOutput			: INT;				// adjusted minimum card count output
					m_rMaxOutput			: INT;				// adjusted maximum card count output *)


(*UPDATE: 			March. 30 2021 - MDC

					Code Ported from Wago. Datatypes in Wago for card links are UINT, in Beckhoff they are INT
					
					Offset in GetZeroCalValue detected if needed for 4-20mA, but not used for 0-10V cards
					
					AO_ChannelOutputs changed to reflect.
					
					Tested on a -10V to 10V card EL4034
*)		
	
(*UPDATE: 			March. 18 2021 - Jaison Schaab

					Code Ported from Wago.
					
					Code has NOT Yet been tested.
*)			

FUNCTION_BLOCK fb_AnalogOutputActuator
VAR_INPUT
	AnalogSignalValue		: REAL;						// Analog Signal Value (4-20 mA)
END_VAR
VAR_OUTPUT
	Channel					: AO_ChannelOutputs;		// Scaled Channel Value (ex. COUNTS)
	rawValue				: REAL;						// Raw Input Value (May be removed)
	zeroCalValue			: REAL;						// Zero Calibration Value
END_VAR
VAR
	m_filter 				: fb_FilterExp;		// exponential weighted filter
	
	m_rFilteredValue		: REAL;				// filtered Value
	
	m_Channel				: REAL;				// Internal Channel Signal
	
// Card input (4 to 20 mA)
	m_rMinInput				: REAL;				// minimum commanded input (4.0 mA command)
	m_rMaxInput				: REAL;				// maximum commanded input (20.0 mA command)

// Card output (counts, -32768 to 32767)
	m_iMinOutput			: INT;				// adjusted minimum card count output
	m_iMaxOutput			: INT;				// adjusted maximum card count output

// Offset for Scaling (For Voltage cards = 0, for 4-20mA cards = 4)	
	m_iOffset				: INT;
	
// Underrange / Wire Break Error Detection
	m_underRangeTON			: TON;				// timer ON
	m_underRangeP			: R_TRIG;			// positive edge detection (set alarm)
	m_underRangeN			: F_TRIG;			// negative edge detection (clear alarm)

// Overrange Error Detection
	m_overRangeTON			: TON;				// timer ON
	m_overRangeP			: R_TRIG;			// positive edge detection (set alarm)
	m_overRangeN			: F_TRIG;			// negative edge detection (clear alarm)

// Error (short circuit)
	m_shortCircuitTON		: TON;      		// timer ON
    m_shortCircuitP			: R_TRIG;			// positive edge detection (set alarm)
    m_shortCircuitN			: F_TRIG;			// negative edge detection (clear alarm)	

// Error (wire break)
	m_errorTON				: TON;      		// timer ON
    m_errorP				: R_TRIG;			// positive edge detection (set alarm)
    m_errorN				: F_TRIG;			// negative edge detection (clear alarm)
	
// Fault Handling (Alarms)
	m_devId					: UDeviceId;		// Device Id used for alarm integration
	m_pAlarmHandler			: POINTER TO fb_AlarmHandler;	// Alarm handler function pointer

// Calibration Handling
	m_zeroCalTimer			: fb_elapseTimer;	// duration timer
	m_zeroCalEnable			: BOOL;				// enable flag for the zero calibration routine
	m_zeroCalRunning		: BOOL;				// TRUE if calibration routine running, FALSE otherwise
	m_zeroCalAccumulator	: REAL;				// accumulator (to calculate the averge value)
	m_zeroCalCounter		: UINT;				// counter (to calculate the average value)
	m_rawVal				: REAL;				// raw filtered before scaling
	
END_VAR

// Filter the input value, Filtering Not Required <GRAHAM>
//m_filter(inputValue:= AnalogSignalValue, filteredValue=> m_rFilteredValue);

// Output the raw value - Convert to INT as this is the precision of the input channel value <JAISON>
//rawValue := TO_INT(m_rFilteredValue);
 
// Scale the raw data value to an output value
// Fixed - April 2 / 2020 - Now using standard scaling function. <JAISON>
Channel.value :=  TO_INT(f_LinearScale	  (value 	 := AnalogSignalValue,
										minInput := m_rMinInput, // Already Real Values
										maxInput := m_rMaxInput,
										minOutput := TO_REAL(m_iMinOutput),
										maxOutput := TO_REAL(m_iMaxOutput)));

//
// Under range fault detection, 
// 
// NOT USED FOR THE 750-563 card but some of this functionality may be used in the future <GRAHAM>


IF (m_zeroCalEnable) THEN	

	// Calibration handling (zeroing) <TODO>
	m_zeroCalTimer();

	// Check if we are currently zeroing the transducer
	IF (m_zeroCalTimer.uliElapsedTime > 0) THEN

		// Update the data values
		m_zeroCalAccumulator := m_zeroCalAccumulator + m_filter.filteredValue;
		m_zeroCalCounter := m_zeroCalCounter + 1;

	ELSE

		// Done, calculate the average value
		IF (m_zeroCalCounter > 0) THEN

			m_rawVal := m_zeroCalAccumulator / m_zeroCalCounter;
	
		ELSE
	
			m_rawVal := m_filter.filteredValue;

		END_IF
		
		m_zeroCalRunning := FALSE;
		
	END_IF

ELSE
	
	// If no calibration is done set value to 0
	m_rawVal := 0;

END_IF

// Scale the raw calibration value to an output value
zeroCalValue := GetZeroCalValue();

(* ---------------------------------------------------------------------------
Func name   : 	AbortCal
Description : 	Aborts the calibration routine
Inputs      :	None
Returns     : 	None
Notes       : 	This routine will 0 out any previous output calibration value
--------------------------------------------------------------------------- *)

METHOD AbortCal
VAR_INPUT
END_VAR
m_zeroCalEnable := FALSE;
m_zeroCalAccumulator := 0.0;
m_zeroCalCounter := 0;
zeroCalValue := 0;
END_METHOD

(* ---------------------------------------------------------------------------
Func name   : 	Arm
Description : 	Enables all assiciated analog output alarms
Inputs      :	devId	-	device Id associated with the alarms in the system
Returns     : 	None
Notes       : 	The local alarm handler pointer is simply points to the
				global alarm handle function block.  Another approach could
				be to have any users of the analog transducer supply a
				fault handling routine with a common interface.
--------------------------------------------------------------------------- *)

METHOD Arm
VAR_INPUT
	devId		: UDeviceId;
END_VAR
// Set the local alarm handler pointer to the global handler so that the fault handler function can set alarms
m_pAlarmHandler := ADR(gAlarmHandler);

// Set the Device Id
m_devId := devId;
END_METHOD

(* ---------------------------------------------------------------------------
Func name   : 	Disarm
Description : 	Disables all assiciated analog output alarms
Inputs      :	None
Returns     : 	None
Notes       : 	This routine will also clear any active alarms before
				disabling the handler.
--------------------------------------------------------------------------- *)

METHOD Disarm
VAR_INPUT
END_VAR
// Clear any active alarms - Is this needed?
Fault(fault:= f_FaultCode(TFaultPriority.Error, TFaultCondition.UnderRange), state:= FALSE);
Fault(fault:= f_FaultCode(TFaultPriority.Error, TFaultCondition.OverRange), state:= FALSE);
Fault(fault:= f_FaultCode(TFaultPriority.Error, TFaultCondition.HwError), state:= FALSE);

// Clear the local alarm handler pointer - This will ignore all calls
m_pAlarmHandler := 0;
END_METHOD

(* ---------------------------------------------------------------------------
Func name   : 	Fault
Description : 	fault handling routine used as a common interface for
				setting/clearing analog output faults.
Inputs      :	fault	-	fault code
				state	-	state of the fault
Returns     : 	None
Notes       : 	This routine assumes that when the transducer is armed,
				the alarm handler pointer will be non-zero, as well the
				internal m_devId parameter is set and valid.
--------------------------------------------------------------------------- *)

METHOD Fault
VAR_INPUT
	fault	: UFaultCode;
	state	: BOOL;
END_VAR
IF (m_pAlarmHandler <> 0) THEN
	
	IF (state) THEN
	
		m_pAlarmHandler^.Set(code:= f_AlarmCode(m_devId, fault));	
	
	ELSE
		
		m_pAlarmHandler^.Clear(code:= f_AlarmCode(m_devId, fault));	
	
	END_IF

END_IF
END_METHOD

(* ---------------------------------------------------------------------------
Func name   : 	FB_exit
Description : 	Destructor
Inputs      :	None
Returns     : 	None
Notes       : 	
--------------------------------------------------------------------------- *)

METHOD FB_exit : BOOL
VAR_INPUT
	bInCopyCode : BOOL; // if TRUE, the exit method is called for exiting an instance that is copied afterwards (online change)
END_VAR
// Do nothing
END_METHOD

(* ---------------------------------------------------------------------------
Func name   : 	FB_init
Description : 	Constructor
Inputs      :	iMinInput			:	minimum input
				iMaxInput			: 	maximum input
				rMinOutput			:	minimum output
				rMaxOutput			:	maximum output
				uiFilterSize 		:	Filter Sample Size
				uiFilterPrecision	:	Filter precision
				tDelay				:	Timer On Delay value
Returns     : 	None
Notes       : 	
--------------------------------------------------------------------------- *)

METHOD FB_init : BOOL
VAR_INPUT
	bInitRetains 				: BOOL; 		// if TRUE, the retain variables are initialized (warm start / cold start)
    bInCopyCode  				: BOOL; 		// if TRUE, the instance afterwards gets moved into the copy code (online change)
	rMinInput					: REAL;			// minimum input
	rMaxInput					: REAL;			// maximum input
	iMinOutput					: INT;			// minimum output
	iMaxOutput					: INT;			// maximum output
END_VAR
// Set the member variables
m_rMinInput 	:= rMinInput;
m_rMaxInput		:= rMaxInput;
m_iMinOutput	:= iMinOutput;
m_iMaxOutput 	:= iMaxOutput;

// Initialize the calibration variables
m_zeroCalTimer.Initialize(msec:= 0, countDown:= TRUE, freeze:= FALSE);
m_zeroCalEnable := FALSE;
m_zeroCalRunning := FALSE;
m_zeroCalAccumulator := 0.0;
m_zeroCalCounter := 0;

// Initialize the 'underrange', 'overrange', and 'error' positive edge detect signals
// to low so that we detect a positive edge if the signal is high at startup.
m_underRangeP(CLK:=FALSE);
m_overRangeP(CLK:=FALSE);
m_errorP(CLK:=FALSE);

// Initialize the output variables
Channel.value := 0;
rawValue := 0;
zeroCalValue := 0;

// Set the local alarm handler pointer to the global handler
m_pAlarmHandler := ADR(gAlarmHandler);
END_METHOD

(* ---------------------------------------------------------------------------
Func name   : 	GetDevId
Description : 	Returns the transducer Device Id used for alarm categorization.
Inputs      :	None
Returns     : 	UDeviceId	-	Transducer device ID variable
Notes       : 	This function is currently used by the ENDP_Analog function block.
				I believe the End Point should set the Device Id instead of getting
				it from the transducer.  This could be a future improvement.
--------------------------------------------------------------------------- *)

METHOD GetDevId : UDeviceId
VAR_INPUT
END_VAR
GetDevId := m_devId;
END_METHOD

(* ---------------------------------------------------------------------------
Func name   : 	GetMaxOutput
Description : 	Returns the maximum output value of the transducer.
Inputs      :	None
Returns     : 	REAL	-	transducer maximum output value
Notes       : 	This routine is used by the fb_ENDP_Analog to get the
				transducer output limits.
--------------------------------------------------------------------------- *)

METHOD PUBLIC GetMaxInput : REAL
VAR_INPUT
END_VAR
GetMaxInput := m_rMaxInput;
END_METHOD

(* ---------------------------------------------------------------------------
Func name   : 	GetMaxOutput
Description : 	Returns the maximum output value of the transducer.
Inputs      :	None
Returns     : 	REAL	-	transducer maximum output value
Notes       : 	This routine is used by the fb_ENDP_Analog to get the
				transducer output limits.
--------------------------------------------------------------------------- *)

METHOD PUBLIC GetMaxOutput : REAL
VAR_INPUT
END_VAR
GetMaxOutput := m_iMaxOutput;
END_METHOD

(* ---------------------------------------------------------------------------
Func name   : 	GetMinOutput
Description : 	Returns the minimum output value of the transducer.
Inputs      :	None
Returns     : 	REAL	-	transducer minimum output value
Notes       : 	This routine is used by the fb_ENDP_Analog to get the
				transducer output limits.
--------------------------------------------------------------------------- *)

METHOD PUBLIC GetMinInput : REAL
VAR_INPUT
END_VAR
GetMinInput := m_rMinInput;
END_METHOD

(* ---------------------------------------------------------------------------
Func name   : 	GetMinOutput
Description : 	Returns the minimum output value of the transducer.
Inputs      :	None
Returns     : 	REAL	-	transducer minimum output value
Notes       : 	This routine is used by the fb_ENDP_Analog to get the
				transducer output limits.
--------------------------------------------------------------------------- *)

METHOD PUBLIC GetMinOutput : REAL
VAR_INPUT
END_VAR
GetMinOutput := m_iMinOutput;
END_METHOD

(* ---------------------------------------------------------------------------
Func name   : 	GetZeroCalValue
Description : 	Scales and returns the current calibration value in mA.
Inputs      :	None
Returns     : 	REAL	-	scaled calibration value (mA)
Notes       : 	
--------------------------------------------------------------------------- *)

METHOD GetZeroCalValue : REAL
VAR_INPUT
END_VAR
VAR
	iOffset : INT;
END_VAR
//Offset detected and used with 4-20 cards, otherwise no offset
IF m_iMinOutput = 4 THEN 
	iOffset := 4;
ELSE
	iOffset := 0;
END_IF

// Scale the raw calibration value to an output value
 GetZeroCalValue := (m_rawVal * (m_iMaxOutput - m_iMinOutput) / (m_rMaxInput - m_rMinInput) + iOffset);
END_METHOD

(* ---------------------------------------------------------------------------
Func name   : 	InitAlarms
Description : 	Initializes the deviceId member variable used to set/clear
				the approproate alarms.
Inputs      :	devId	:	Device Id used for alarm integration
Returns     : 	None
Notes       : 	
--------------------------------------------------------------------------- *)

METHOD InitAlarms
VAR_INPUT
	devId		: UDeviceId;	// Device Id used for alarm integration
END_VAR
// Set the device id which is used for alarm integrtion
m_devId := devId;

// Register the handled alarm codes
m_pAlarmHandler^.RegisterAlarmCode(f_AlarmCode(m_devId, f_FaultCode(TFaultPriority.Error, TFaultCondition.UnderRange)));
m_pAlarmHandler^.RegisterAlarmCode(f_AlarmCode(m_devId, f_FaultCode(TFaultPriority.Error, TFaultCondition.OverRange)));
m_pAlarmHandler^.RegisterAlarmCode(f_AlarmCode(m_devId, f_FaultCode(TFaultPriority.Error, TFaultCondition.ShortCircuit)));
m_pAlarmHandler^.RegisterAlarmCode(f_AlarmCode(m_devId, f_FaultCode(TFaultPriority.Error, TFaultCondition.HwError)));
END_METHOD

(* ---------------------------------------------------------------------------
Func name   : 	IsZeroCalRunning
Description : 	Returns the status of the zero cal routine.
Inputs      :	None
Returns     : 	TRUE if zero cal running, FALSE otherwise
Notes       : 	
--------------------------------------------------------------------------- *)

METHOD IsZeroCalRunning : BOOL
VAR_INPUT
END_VAR
IsZeroCalRunning := m_zeroCalRunning;
END_METHOD

(* ---------------------------------------------------------------------------
Func name   : 	ZeroCal
Description : 	Averages the transducer signal input value to provide
				a calibration value reresenting a zero offset
Inputs      :	duration_ms	-	Duration of value averaging time in ms
Returns     : 	None
Notes       : 	This initializes the timer which runs the averaging routine
				in the main function block instantiation code.
--------------------------------------------------------------------------- *)

METHOD ZeroCal
VAR_INPUT
	duration_ms		: UINT;
END_VAR
// Initialize the data
m_zeroCalTimer.Initialize(msec := duration_ms, countDown := TRUE, freeze := FALSE);
m_zeroCalEnable := true;
m_zeroCalAccumulator := 0.0;
m_zeroCalCounter := 0;
zeroCalValue := 0;
m_zeroCalRunning := TRUE;
END_METHOD

END_FUNCTION_BLOCK

// 20 Program Organization Units/Utility Functions/f_LinearScale
(*AUTHOR:			Jaison Schaab*)
(*DATE:				April 2 / 2020*)
(*DESCRIPTION: 		This Function will generate a linear scaled value based on the input limits.
					Using this function for all scaling will standardize scaling throughout the
					library. *)

(*UPDATE: 			March. 22 2021 - Jaison Schaab

					Code Is fully tested and functional.
					
*)

(*UPDATE: 			March. 18 2021 - Jaison Schaab

					Code Ported from Wago.
					
					Code has NOT Yet been tested.
*)
				
(*UPDATE: 			June. 9 2020 - Jaison Schaab

					Added error checking to ensue the m_slope divisor was NOT 0.
*)
				
FUNCTION f_LinearScale : REAL
VAR_INPUT
	value			: REAL;		// input value
	minInput		: REAL;		// minimum input value
	maxInput		: REAL;		// maximum input value
	minOutput		: REAL;		// minimum output value
	maxOutput		: REAL;		// maximum output value
END_VAR
VAR
	m_slope			: REAL;		// scale slope
	m_offset		: REAL;		// scale offset
END_VAR

IF (ABS(maxInput - minInput) > 0) THEN
	
	// Calculate the slope - m
	m_slope := (maxOutput - minOutput) / (maxInput - minInput);

	// Calculate the offset - b
	m_offset := minOutput - (m_slope * minInput);

	// Calculate the scaled value - y = mx + b
	f_LinearScale := (value * m_slope) + m_offset;
	
ELSE
	
	f_LinearScale := 0;
	
END_IF

END_FUNCTION

// 20 Program Organization Units/Utility Functions/fb_FilterExp
(*AUTHOR:			Jaison Schaab*)
(*DATE:				November 20 / 2019*)
(*DESCRIPTION: 		The following exponential filter will achieve approximately 
*					63.2% of a step input by the specified sample size. *)

(*UPDATE: 			March. 22 2021 - Jaison Schaab

					Code Is fully tested and functional.				
*)

(*UPDATE: 			March. 18 2021 - Jaison Schaab

					Code Ported from Wago.
					
					Code has NOT Yet been tested.
*)

FUNCTION_BLOCK fb_FilterExp
VAR_INPUT
	inputValue			: REAL := 0;	// Input Value
END_VAR
VAR_OUTPUT
	filteredValue		: REAL;			// Filtered Value
END_VAR
VAR
	m_sampleSize		: UINT;			// Filter Sample Size
	m_precision			: UINT;			// Filter precision
    m_expWtFactor		: REAL;			// Exponential Weight Factor
	m_digitsToTruncate	: REAL;			// Number of digits (base 10) to truncate
	m_movingAverage		: REAL := 0;	// Filtered Value
END_VAR
VAR CONSTANT
	m_exp				: INT := -1;	// must not be zero
END_VAR

// Keep the history of the previous values in 'movingAverage'
m_movingAverage := m_movingAverage + (m_expWtFactor * (inputValue - m_movingAverage));

// Output the filtered value
// Truncate filtered value so we do not experience "infinite" decline approaching 0}
filteredValue := DINT_TO_REAL(REAL_TO_DINT(m_movingAverage * m_digitsToTruncate)) / m_digitsToTruncate;

(* ---------------------------------------------------------------------------
Func name   : 	FB_exit
Description : 	Destructor
Inputs      :	None
Returns     : 	None
Notes       : 	
--------------------------------------------------------------------------- *)

METHOD FB_exit : BOOL
VAR_INPUT
	bInCopyCode : BOOL; // if TRUE, the exit method is called for exiting an instance that is copied afterwards (online change)
END_VAR
// Do nothing
END_METHOD

(* ---------------------------------------------------------------------------
Func name   : 	FB_init
Description : 	Constructor
Inputs      :	None
Returns     : 	None
Notes       : 	No parameters are required. Use initialize() routine
				to setup analog transducer.
--------------------------------------------------------------------------- *)

METHOD FB_init : BOOL
VAR_INPUT
	bInitRetains 		: BOOL; 		// if TRUE, the retain variables are initialized (warm start / cold start)
    bInCopyCode  		: BOOL; 		// if TRUE, the instance afterwards gets moved into the copy code (online change)
END_VAR
VAR CONSTANT
	DEFAULT_SAMPLE_SIZE	: UINT	:= 10;	// Filter Sample Size, this value will be overwritten by the "initialize" method
	DEFAULT_PRECISION	: UINT	:= 4;	// Filter precision, this value will be overwritten by the "initialize" method
END_VAR
// Set a default value for the sample size, This value will be overwritten by the "initialize" method
m_sampleSize := DEFAULT_SAMPLE_SIZE;

// Set a default value for the precision, This value will be overwritten by the "initialize" method
m_precision := DEFAULT_PRECISION;

// Exponential weight factor should be less than 1 and as a guideline
// weight = number of samples ^ -1
m_expWtFactor := LREAL_TO_REAL(EXPT(MAX(m_sampleSize, 1), m_exp)); 

// Calculate the number of digits (base 10) to truncate
m_digitsToTruncate := LREAL_TO_REAL(EXPT(10.0, m_precision));

// Initialize the filtered value
m_movingAverage := 0;
END_METHOD

(* ---------------------------------------------------------------------------
Func name   : 	GetSampleSize
Description : 	retrieves the filter sample size paramter
Inputs      :	None
Returns     : 	UINT	- current filter sample size
Notes       : 	
--------------------------------------------------------------------------- *)

METHOD GetSampleSize : UINT
VAR_INPUT
END_VAR
GetSampleSize := DINT_TO_UINT(TRUNC(EXPT(10, LOG(m_expWtFactor)/m_exp)));
END_METHOD

(* ---------------------------------------------------------------------------
Func name   : 	Initialize
Description : 	initializes the filters parameters
Inputs      :	sampleSize	- sample size of the filter
				precision	- value precision of the filter output	
Returns     : 	None
Notes       : 	
--------------------------------------------------------------------------- *)

METHOD Initialize
VAR_INPUT
	sampleSize			: UINT;			// Filter Sample Size - Value of 0 or 1 will disable the filter <JAISON>
	precision			: UINT;			// Filter precision
END_VAR
// Set the default value for the sample size
m_sampleSize := sampleSize;

// Set the default value for the precision
m_precision := precision;

// Exponential weight factor should be less than 1 and as a guideline
// weight = number of samples ^ -1
m_expWtFactor := LREAL_TO_REAL(EXPT(MAX(m_sampleSize, 1), m_exp)); 

// Calculate the number of digits (base 10) to truncate
m_digitsToTruncate := LREAL_TO_REAL(EXPT(10.0, m_precision));

// Initialize the filtered value
m_movingAverage := 0;
END_METHOD

(* ---------------------------------------------------------------------------
Func name   : 	SetSampleSize
Description : 	sets the filter sample size parameter
Inputs      :	size	- desired filter sample size
Returns     : 	BOOL	- TRUE on success, else FALSE
Notes       : 	
--------------------------------------------------------------------------- *)

METHOD SetSampleSize : BOOL
VAR_INPUT
	size	: UINT;
END_VAR
m_sampleSize := size;

// Exponential weight factor should be less than 1 and as a guideline
// weight = number of samples ^ -1
m_expWtFactor := LREAL_TO_REAL(EXPT(MAX(m_sampleSize, 1), m_exp)); 

// Return True
SetSampleSize := TRUE;
END_METHOD

END_FUNCTION_BLOCK

// 20 Program Organization Units/Utility Functions/fb_ElapseTimer
(*AUTHOR:			Jaison Schaab*)
(*DATE:				November 20 / 2019*)
(*DESCRIPTION: 		The following elapse timer function block will count up or down
*					a specified duration in milliseconds based on initialization parameters. *)

(*UPDATE: 			March. 22 2021 - Jaison Schaab

					Code Is fully tested and functional.				
*)

(*UPDATE: 			March. 18 2021 - Jaison Schaab

					Code Ported from Wago.
					
					Code has NOT Yet been tested.
*)

FUNCTION_BLOCK fb_ElapseTimer
VAR_INPUT
END_VAR
VAR_OUTPUT
	uliElapsedTime	: ULINT;		// current elapsed time in msec
END_VAR
VAR
	m_elapse		: ULINT;		// elapse time, in msec
	m_ref			: ULINT;		// reference time, in msec

	m_time			: ULINT;		// start time, in msec
	m_countDown		: BOOL;			// true = count down, false = count up
	m_frozen		: BOOL;			// true = frozen
	
	lap				: ULINT;		// lap time, in msec
	diff			: ULINT;		// time difference, in msec
END_VAR
VAR CONSTANT
	maximum			: ULINT := INT_TO_ULINT(-1);	// maximum ULINT value
END_VAR

IF (m_frozen = FALSE) THEN

	// Get the end time (in ms).
	lap := TIME_TO_ULINT(TIME());

	// Calculate the elapsed time and check if it has wrapped around to zero.
	IF (lap >= m_ref) THEN
		
		diff := lap - m_ref;
		
	ELSE
		
		diff := lap + (maximum - m_ref + 1);
			
	END_IF

	// Adjust the timeout value.
	IF (m_countDown) THEN

		m_elapse := SEL(m_elapse > diff, 0, m_elapse - diff);
		
	ELSE

		m_elapse := SEL((m_elapse - m_time) > (m_time - diff), m_elapse + diff, m_time);
			
	END_IF

	// Update the reference time to the last time value.
	m_ref := lap;
	
END_IF

// Return the elapse time, in msec
uliElapsedTime := SEL(m_countDown, m_elapse - m_time, m_elapse);

(* ---------------------------------------------------------------------------
Func name   : 	FB_exit
Description : 	Destructor
Inputs      :	None
Returns     : 	None
Notes       : 	
--------------------------------------------------------------------------- *)

METHOD FB_exit
VAR_INPUT
	bInCopyCode : BOOL; // if TRUE, the exit method is called for exiting an instance that is copied afterwards (online change)
END_VAR
// Do nothing
END_METHOD

(* ---------------------------------------------------------------------------
Func name   : 	FB_init
Description : 	Constructor
Inputs      :	None
Returns     : 	None
Notes       : 	
--------------------------------------------------------------------------- *)

METHOD FB_init
VAR_INPUT
	bInitRetains 		: BOOL; 			// if TRUE, the retain variables are initialized (warm start / cold start)
    bInCopyCode  		: BOOL; 			// if TRUE, the instance afterwards gets moved into the copy code (online change)
END_VAR
VAR CONSTANT
	DEFAULT_START_TIME	: ULINT := 0;		// start time, in msec, this value will be overwritten by the "initialize" method
	DEFAULT_COUNTDOWN	: BOOL := TRUE;		// true = count down, false = count up, this value will be overwritten by the "initialize" method
	DEFAULT_FREEZE		: BOOL := FALSE;	// true = frozen, this value will be overwritten by the "initialize" method
END_VAR
m_time := DEFAULT_START_TIME;
m_countDown := DEFAULT_COUNTDOWN;
m_frozen := DEFAULT_FREEZE;

Reset();
END_METHOD

(* ---------------------------------------------------------------------------
Func name   : 	Freeze
Description : 	updates the blocks frozen flag which will either freeze or
				unfrezzed the elapse timer
Inputs      :	frozen	-	desired state of the frozen flag
Returns     : 	None
Notes       : 	
--------------------------------------------------------------------------- *)

METHOD Freeze
VAR_INPUT
	frozen	: BOOL;
END_VAR
IF(frozen <> m_frozen) THEN
	
	IF(frozen = FALSE) THEN

		// Reset the reference time (in ms).
		m_ref := TIME_TO_ULINT(TIME());
		
	END_IF
	
	m_frozen := frozen;
	
END_IF
END_METHOD

(* ---------------------------------------------------------------------------
Func name   : 	Initialize
Description : 	initializes the timer parameters, starts the timer operation
Inputs      :	msec		- timer duration value in milliseconds
				countDown	- desired timer operation, TRUE = count down, FALSE = count up	
				freeze		- desired state of the frozen flag
Returns     : 	None
Notes       : 	
--------------------------------------------------------------------------- *)

METHOD Initialize
VAR_INPUT
	msec				: ULINT := 0;		// start time, in msec
	countDown			: BOOL := TRUE;		// true = count down, false = count up
	freeze				: BOOL := FALSE;	// true = frozen
END_VAR
m_time := msec;
m_countDown := countDown;
m_frozen := freeze;

Reset();
END_METHOD

(* ---------------------------------------------------------------------------
Func name   : 	Freeze
Description : 	resets the timer parameters to restart timer operation
Inputs      :	None
Returns     : 	None
Notes       : 	
--------------------------------------------------------------------------- *)

METHOD Reset
VAR_INPUT
END_VAR
m_elapse	:= m_time;    				// elapse time, in ms
m_ref		:= TIME_TO_ULINT(TIME()); 	// reference time (in ms)
END_METHOD

END_FUNCTION_BLOCK

// 20 Program Organization Units/Instrument-Controller Functions/fb_ENDP_Analog
(*UPDATE: 			April. 28 2020 - Jaison Schaab

					Added the InitAlarms function which now NEEDS to be called in order to properly hook up the alarm monitors.
					This method is required because codesys does NOT properly propogate the FB_Init information like constructors
					in C code, so it is impossible to pass down the devceId information.
*)

(*UPDATE: 			March. 22 2021 - Jaison Schaab

					Code Is fully tested and functional.	
*)

(*UPDATE: 			March. 18 2021 - Jaison Schaab

					Code Ported from Wago.
					
					Code has NOT Yet been tested.
*)

FUNCTION_BLOCK fb_ENDP_Analog
VAR_INPUT
	//input_Mamp : REAL; use P_TO to get value in Hz. It will be already filtered thru HistAvg(10,2)
END_VAR
VAR_OUTPUT
	physValue : REAL;
	endpState : INT;
END_VAR
VAR
	m_pTxducer420 : POINTER TO fb_AnalogTransducer;
	m_inMin : REAL;
	m_inMax : REAL;
	m_outMin : REAL;
	m_outMax : REAL;
	m_inpdiffDivisor : REAL;
	m_offset : REAL;
	m_hysteresis : REAL;
	//this is all alarm-related down from here. Should be separated into Alarmable interface, if possible.
	m_devId					: UDeviceId;			// Device Id used for alarm integration
	//m_pAlarmHandler : POINTER TO fb_AlarmHandler; //Alarm handler function pointer
	LowAlarmMonitor : fb_AlarmMonitor;
	LowWarningMonitor : fb_AlarmMonitor;
	HighWarningMonitor : fb_AlarmMonitor;
	HighAlarmMonitor : fb_AlarmMonitor;
END_VAR
VAR CONSTANT
	DELAY_TON	: TIME := T#200MS;	//AlarmMonitor delay for Value to DEFINITEVILY cross the alarm limit boundary. and then Trigger.
END_VAR

//get transducers Value scaled from 4_20 to Physical  
physValue := Scale(m_pTxducer420^.signalValue);
//Monitor alarms.
LowAlarmMonitor.MonitorReal(physValue);
LowWarningMonitor.MonitorReal(physValue);
HighWarningMonitor.MonitorReal(physValue);
HighAlarmMonitor.MonitorReal(physValue);

//ALSO_ update the so-called GaugeState. It controls Needle-Color. BY-DESIGN HW-Error also paints Needle in RED.
IF (m_pTxducer420^.channel.error) THEN
	endpState := TEnuHmiGaugeState.LowAlarm;
ELSIF(HighAlarmMonitor.GetState()) THEN
	endpState := TEnuHmiGaugeState.HighAlarm;
ELSIF(LowAlarmMonitor.GetState()) THEN
	endpState := TEnuHmiGaugeState.LowAlarm;
ELSIF(HighWarningMonitor.GetState()) THEN
	endpState := TO_INT(TEnuHmiGaugeState.HighWarning);
ELSIF(LowWarningMonitor.GetState()) THEN
	endpState := TEnuHmiGaugeState.LowWarning;
ELSE
	endpState := TEnuHmiGaugeState.No_Alarm;			
END_IF

(* ---------------------------------------------------------------------------
Func name   : 	FB_init
Description : 	ENDP_Analog_Txducer
Inputs      :	2 reals - are a Range of phys.values sensor is spec-ed to.  
                pointer to fb_Txducer reading the freq.card inputs
Returns     : 	None
--------------------------------------------------------------------------- *)

METHOD FB_init : BOOL
VAR_INPUT
	bInitRetains 		: BOOL; 		// if TRUE, the retain variables are initialized (warm start / cold start)
    bInCopyCode  		: BOOL; 		// if TRUE, the instance afterwards gets moved into the copy code (online change)
	
	ptrTxducer : POINTER TO fb_AnalogTransducer;
	physMin : REAL;
	physMax : REAL;
	perctHysteresis : REAL;
END_VAR
m_pTxducer420 := ptrTxducer;
m_inMin := m_pTxducer420^.GetMinOutput();
m_inMax := m_pTxducer420^.GetMaxOutput();
m_outMin := physMin;    //these are the range of physical values, metric - kPa kg etc
m_outMax := physMax;    //that 4-20 transducer is scaled to.
m_inpdiffDivisor := (m_inMax - m_inMin);
IF (0.0 = m_inpdiffDivisor) THEN
	m_inpdiffDivisor := 0.000001; //protect against div-by-0, only ONCE, and produce VERY-LARGE Bad value.
                                  //Beckhoff-tcNov was doing this A.every cycle and B.returned 0.0 if Bad, which is normal value. hard to notice.
END_IF

//m_pAlarmHandler := ADR(gAlarmHandler); //i am no longer handling Alarms myself. AlarmMonitor does interfacing to 'gAlarmHandler'.
//m_devId := m_pTxducer420^.GetDevId();

m_hysteresis := perctHysteresis/100;
//LowAlarmMonitor.Init(f_AlarmCode(m_devId, f_FaultCode(TFaultPriority.Warning, TFaultCondition.UnderLimit)), TAlarmMonitorType.lower_limit, DELAY_TON);
//LowWarningMonitor.Init(f_AlarmCode(m_devId, f_FaultCode(TFaultPriority.Warning, TFaultCondition.UnderWarning)), TAlarmMonitorType.lower_limit, DELAY_TON);
//HighWarningMonitor.Init(f_AlarmCode(m_devId, f_FaultCode(TFaultPriority.Warning, TFaultCondition.OverWarning)), TAlarmMonitorType.upper_limit, DELAY_TON);
//HighAlarmMonitor.Init(f_AlarmCode(m_devId, f_FaultCode(TFaultPriority.Warning, TFaultCondition.OverLimit)), TAlarmMonitorType.upper_limit, DELAY_TON);
END_METHOD

METHOD Get_UserAlarms
VAR_OUTPUT
	outLAlarm : REAL;
	outLWarn : REAL;
	outHWArn : REAL;
	outHAlarm : REAL;
END_VAR
outLAlarm := LREAL_TO_REAL(LowAlarmMonitor.m_limit.limitOn);
outLWarn  := LREAL_TO_REAL(LowWarningMonitor.m_limit.limitOn);
outHWArn  := LREAL_TO_REAL(HighWarningMonitor.m_limit.limitOn);
outHAlarm := LREAL_TO_REAL(HighAlarmMonitor.m_limit.limitOn);
END_METHOD

(* ---------------------------------------------------------------------------
Func name   : 	GetConfigData
Description : 	equivalent of "Configure" bkhff-legacy-names.
				
Inputs      :	2-end-range-values, 1 offset, 4 alarms - 7 values.
				state	-	state of the fault
Returns     : 	None
Notes       : 	
--------------------------------------------------------------------------- *)

METHOD GetConfigData
VAR_INPUT
	//cfg : TEndpAnalogCfg;
MinValue : REAL;
MaxValue : REAL;
OffsetValue : REAL;
LowLimit : REAL;
LowWarning : REAL;
HighWarning : REAL;
HighLimit : REAL;
END_VAR
m_outMin := MinValue;
m_outMax := MaxValue;
m_offset := OffsetValue;

//LowAlarmMonitor.m_limit.limitOn := LowLimit;
LowAlarmMonitor.SetLimitReal(LowLimit, LowLimit*(1 + m_hysteresis)); // + 0.5);

//LowWarningMonitor.m_limit.limitOn := LowWarning;
LowWarningMonitor.SetLimitReal(LowWarning, LowWarning*(1 + m_hysteresis)); // + 0.5);

//HighWarningMonitor.m_limit.limitOn := HighWarning;
HighWarningMonitor.SetLimitReal(HighWarning, HighWarning*(1 - m_hysteresis)); // - 0.5);

//HighAlarmMonitor.m_limit.limitOn := HighLimit;
HighAlarmMonitor.SetLimitReal(HighLimit, HighLimit*(1 - m_hysteresis)); // - 0.5);
END_METHOD

METHOD GetRange_MinMax
VAR_OUTPUT
	outMinVal : REAL;
	outMaxVal : REAL;
END_VAR
// these are the ENDP product values, in physical Units
outMinVal := m_outMin;
outMaxVal := m_outMax;
END_METHOD

(* ---------------------------------------------------------------------------
Func name   : 	InitAlarms
Description : 	Initializes the deviceId member variable and all alarm
				monitors.
Inputs      :	None
Returns     : 	None
Notes       : 	This needs to be called AFTER the transducer alarms are
				initialized.
--------------------------------------------------------------------------- *)

METHOD InitAlarms
VAR_INPUT
END_VAR
m_devId := m_pTxducer420^.GetDevId();

LowAlarmMonitor.InitAlarm(f_AlarmCode(m_devId, f_FaultCode(TFaultPriority.Warning, TFaultCondition.UnderLimit)), TAlarmMonitorType.lower_limit, DELAY_TON);
LowWarningMonitor.InitAlarm(f_AlarmCode(m_devId, f_FaultCode(TFaultPriority.Warning, TFaultCondition.UnderWarning)), TAlarmMonitorType.lower_limit, DELAY_TON);
HighWarningMonitor.InitAlarm(f_AlarmCode(m_devId, f_FaultCode(TFaultPriority.Warning, TFaultCondition.OverWarning)), TAlarmMonitorType.upper_limit, DELAY_TON);
HighAlarmMonitor.InitAlarm(f_AlarmCode(m_devId, f_FaultCode(TFaultPriority.Warning, TFaultCondition.OverLimit)), TAlarmMonitorType.upper_limit, DELAY_TON);
END_METHOD

METHOD Scale : REAL
VAR_INPUT
	val_mamp : REAL;
END_VAR
Scale := (val_mamp - m_inMin)*(m_outMax - m_outMin)/m_inpdiffDivisor + m_outMin;
END_METHOD

METHOD Set_Hysteresis
VAR_INPUT
	perctHysteresis : REAL;
END_VAR
m_hysteresis := perctHysteresis/100;
END_METHOD

METHOD SetRange_MinMax
VAR_INPUT
	physMin : REAL;
	physMax : REAL;
END_VAR
// these are the ENDP product values, in physical Units
m_outMin := physMin;
m_outMax := physMax;
END_METHOD

METHOD SetRange_UserAlarms
VAR_INPUT
	loAlarm : REAL;
	loWarn : REAL;
	hiWarn : REAL;
	hiAlarm : REAL;
END_VAR
IF (NOTUSED = loAlarm OR NOTUSED_LOMAX = loAlarm OR loAlarm < m_outMin OR loAlarm > m_outMax) THEN
	loAlarm := NOTUSED_LOMAX;
	LowAlarmMonitor.DisableLimit();
ELSE
	LowAlarmMonitor.EnableLimit();
END_IF
LowAlarmMonitor.SetLimitReal(loAlarm, (loAlarm  + MAX(0.001, ABS(loAlarm)) * m_hysteresis));

IF (NOTUSED = loWarn OR loWarn <= loAlarm OR loAlarm > m_outMax) THEN
	loWarn := loAlarm;
	LowWarningMonitor.DisableLimit();
ELSE
	LowWarningMonitor.EnableLimit();
END_IF
LowWarningMonitor.SetLimitReal(loWarn, (loWarn  + MAX(0.001, ABS(loWarn)) * m_hysteresis));

IF (NOTUSED = hiAlarm OR NOTUSED_HIMAX = hiAlarm OR hiAlarm < m_outMin OR hiAlarm > m_outMax) THEN
	hiAlarm := NOTUSED_HIMAX; //Guaranteed greater than m_outMax; We pick _some_ large value.
	HighAlarmMonitor.DisableLimit();
ELSE
	HighAlarmMonitor.EnableLimit();
END_IF
HighAlarmMonitor.SetLimitReal(hiAlarm, (hiAlarm - MAX(0.001, ABS(hiAlarm)) * m_hysteresis));

IF (NOTUSED = hiWarn OR hiWarn >= hiAlarm OR hiWarn < m_outMin) THEN
	hiWarn := hiAlarm;   //User doesnt have ability to set these individually. So WE define this order. So hiAlarm - already set.
	HighWarningMonitor.DisableLimit();
ELSE
	HighWarningMonitor.EnableLimit();
END_IF
HighWarningMonitor.SetLimitReal(hiWarn, (hiWarn - MAX(0.001, ABS(hiWarn)) * m_hysteresis));
END_METHOD

END_FUNCTION_BLOCK

// 20 Program Organization Units/Input-Output Functions/fb_AnalogTransducer
(*AUTHOR:			Jaison Schaab*)
(*DATE:				November 20 / 2019*)
(*DESCRIPTION: 		This Function Block provides a base class for all analog input values.  The block
					will generate a linear scaled value and generate the associated hardware level alarms.
					
					Use the "AI_ChannelInputs" data type to link the channel data from the physical I/O card. *)

(*UPDATE: 			March. 22 2021 - Jaison Schaab

					Code Is fully tested and functional.		
*)

(*UPDATE: 			March. 18 2021 - Jaison Schaab

					Code Ported from Wago.
					
					Code has NOT Yet been tested.
*)
	
(*UPDATE: 			August. 31 2020 - Jaison Schaab

					Moved the ZeroCal calculation to its own "GetZeroCalValue()" Method and added the "m_zeroCalRunning" BOOL with
					matching "IsZeroCalRunning()" Method; this will allow endpoints using the scale routine can determine when 
					the calibration routine is running or not.
*)	
				
(*UPDATE: 			March. 31 2020 - Jaison Schaab

					Added fault handling for the short circuit error which can be generated by certain 
					analog input cards.  Initially designed with the 750-464/040-000 card driver development.
*)

(*UPDATE: 			April. 2 2020 - Jaison Schaab

					Fixed the scaling routine to now use a standard scaling function.  This will ensure
					all linear scaling throughout programs is consistent.
*)

(*UPDATE: 			April. 28 2020 - Jaison Schaab

					Added the InitAlarms function which now NEEDS to be called in order to properly hook up the alarm monitors.
					This method is required because codesys does NOT properly propogate the FB_Init information like constructors
					in C code, so it is impossible to pass down the devceId information.
*)

(*UPDATE: 			June. 23 2020 - Jaison Schaab

					Added "m_pAlarmHandler^.RegisterAlarmCode" function calls in the InitAlarms Method which is required to
					populate the registered alarm code lists in the fb_AlarmHandler class.  The alarms handled by this class
					are:
					
						- f_FaultCode(TFaultPriority.Error, TFaultCondition.UnderRange)
						- f_FaultCode(TFaultPriority.Error, TFaultCondition.OverRange)
						- f_AlarmCode(m_devId, f_FaultCode(TFaultPriority.Error, TFaultCondition.ShortCircuit)
						- f_AlarmCode(m_devId, f_FaultCode(TFaultPriority.Error, TFaultCondition.HwError)
*)	

FUNCTION_BLOCK fb_AnalogTransducer
VAR_INPUT
	channel					: AI_ChannelInputs;	// Input Channel
END_VAR
VAR_OUTPUT
	signalValue				: REAL;				// Scaled Signal Value (ex. mA or VDC)
	rawValue				: REAL;				// Raw Input Value (May be removed)
	zeroCalValue			: REAL;				// Zero Calibration Value
END_VAR
VAR
	m_filter 				: fb_FilterExp;		// exponential weighted filter
	
	m_rFilteredValue		: REAL;				// filtered Value
	
// Transducer input
	m_iMinInput				: INT;				// minimum input
	m_iMaxInput				: INT;				// maximum input

// Transducer output
	m_rMinOutput			: REAL;				// adjusted minimum output
	m_rMaxOutput			: REAL;				// adjusted maximum output
	
// Underrange / Wire Break Error Detection
	m_underRangeTON			: TON;				// timer ON
	m_underRangeP			: R_TRIG;			// positive edge detection (set alarm)
	m_underRangeN			: F_TRIG;			// negative edge detection (clear alarm)

// Overrange Error Detection
	m_overRangeTON			: TON;				// timer ON
	m_overRangeP			: R_TRIG;			// positive edge detection (set alarm)
	m_overRangeN			: F_TRIG;			// negative edge detection (clear alarm)

// Error (short circuit)
	m_shortCircuitTON		: TON;      		// timer ON
    m_shortCircuitP			: R_TRIG;			// positive edge detection (set alarm)
    m_shortCircuitN			: F_TRIG;			// negative edge detection (clear alarm)	

// Error (wire break)
	m_errorTON				: TON;      		// timer ON
    m_errorP				: R_TRIG;			// positive edge detection (set alarm)
    m_errorN				: F_TRIG;			// negative edge detection (clear alarm)
	m_WireBreakDetected		: BOOL;				// TRUE - Wire Break , FALSE - No Wire Break
// Fault Handling (Alarms)
	m_devId					: UDeviceId;		// Device Id used for alarm integration
	m_pAlarmHandler			: POINTER TO fb_AlarmHandler;	// Alarm handler function pointer

// Calibration Handling
	m_zeroCalTimer			: fb_elapseTimer;	// duration timer
	m_zeroCalEnable			: BOOL;				// enable flag for the zero calibration routine
	m_zeroCalRunning		: BOOL;				// TRUE if calibration routine running, FALSE otherwise
	m_zeroCalAccumulator	: REAL;				// accumulator (to calculate the averge value)
	m_zeroCalCounter		: UINT;				// counter (to calculate the average value)
	m_rawVal				: REAL;				// raw filtered before scaling
	
END_VAR

// Filter the input value
m_filter(inputValue:= channel.value, filteredValue=> m_rFilteredValue);

// Output the raw value - Convert to INT as this is the precision of the input channel value <JAISON>
rawValue := TO_INT(m_rFilteredValue);
 
// Scale the raw data value to an output value
// Fixed - April 2 / 2020 - Now using standard scaling function. <JAISON>
signalValue := f_LinearScale(	value := rawValue,
								minInput := TO_REAL(m_iMinInput),
								maxInput := TO_REAL(m_iMaxInput),
								minOutput := m_rMinOutput,
								maxOutput := m_rMaxOutput);

//
// Under range fault detection
//

// Use a TON delay timer - Added condition to ignore underrange if channel error is detected. <JAISON>
m_underRangeTON(IN:= (channel.underRange AND NOT channel.error));

// Rising Edge Trigger
m_underRangeP(CLK:= m_underRangeTON.Q);

// Falling Edge Trigger
m_underRangeN(CLK:= m_underRangeTON.Q);

